// TIA Portal V17 program export: 9 tag tables, 0 data types, 25 data blocks, 98 code blocks (in call order from the OBs), 18 instance data blocks

VAR_GLOBAL   // PLC tag table "AIQ"
   IW100 AT %IW100 : Int;
   IW102 AT %IW102 : Int;
   IW104 AT %IW104 : Int;
   IW106 AT %IW106 : Int;
   IW108 AT %IW108 : Int;
   IW110 AT %IW110 : Int;
   IW112 AT %IW112 : Int;
   IW116 AT %IW116 : Int;
   IW118 AT %IW118 : Int;
   IW120 AT %IW120 : Int;
   IW122 AT %IW122 : Int;
   IW124 AT %IW124 : Int;
   IW126 AT %IW126 : Int;
   IW128 AT %IW128 : Int;
   IW130 AT %IW130 : Int;
   IW132 AT %IW132 : Int;
   IW134 AT %IW134 : Int;
   IW136 AT %IW136 : Int;
   IW138 AT %IW138 : Int;
   IW140 AT %IW140 : Int;
   IW142 AT %IW142 : Int;
   QW100 AT %QW100 : Int;
   QW102 AT %QW102 : Int;
   QW104 AT %QW104 : Int;
   QW106 AT %QW106 : Int;
   QW108 AT %QW108 : Int;
   QW110 AT %QW110 : Int;
   QW112 AT %QW112 : Int;
   QW114 AT %QW114 : Int;
   QW116 AT %QW116 : Int;
   QW118 AT %QW118 : Int;
   QW120 AT %QW120 : Int;
   QW122 AT %QW122 : Int;
   QW124 AT %QW124 : Int;
   QW126 AT %QW126 : Int;
   QW128 AT %QW128 : Int;
   QW130 AT %QW130 : Int;
   QW132 AT %QW132 : Int;
   QW134 AT %QW134 : Int;
   QW136 AT %QW136 : Int;
   QW138 AT %QW138 : Int;
   QW140 AT %QW140 : Int;
   QW142 AT %QW142 : Int;
   QW144 AT %QW144 : Int;
   QW146 AT %QW146 : Int;
   QW148 AT %QW148 : Int;
   QW150 AT %QW150 : Int;
   IW114 AT %IW114 : Int;
   IW144 AT %IW144 : Int;
   IW146 AT %IW146 : Int;
   IW148 AT %IW148 : Int;
   IW150 AT %IW150 : Int;
   IW152 AT %IW152 : Int;
   IW154 AT %IW154 : Int;
   IW156 AT %IW156 : Int;
   IW158 AT %IW158 : Int;
   IW160 AT %IW160 : Int;
   IW162 AT %IW162 : Int;
END_VAR

VAR_GLOBAL   // PLC tag table "AIQM"
   IWJF进风流量计 AT %MW600 : Int;
   IWJL进料流量 AT %MW602 : Int;
   IWJF进风压差变送器 AT %MW604 : Int;
   IWCF出风高效压差变送器 AT %MW606 : Int;
   IWBD布袋压差变送器 AT %MW608 : Int;
   IWSS输送高效压差变送器 AT %MW610 : Int;
   IWJL进料压力 AT %MW612 : Int;
   IWTN塔内压力 AT %MW614 : Int;
   IWGD管道压力变送器 AT %MW616 : Int;
   IWJD进氮压力 AT %MW618 : Int;
   IWFK放空比例反馈 AT %MW620 : Int;
   IWJF进风加热比例反馈 AT %MW622 : Int;
   IWHF回风加热比例反馈 AT %MW624 : Int;
   IWWH雾化油压 AT %MW626 : Int;
   IWYH氧含仪1 AT %MW628 : Int;
   IWYH氧含仪2 AT %MW630 : Int;
   IWYJ一级溶剂液位计 AT %MW632 : Int;
   IWEJ二级溶剂液位计 AT %MW634 : Int;
   IWCW除雾溶剂液位计 AT %MW636 : Int;
   IWSF送风机 AT %MW638 : Int;
   IWYF引风机 AT %MW640 : Int;
   IWLX离心雾化器 AT %MW642 : Int;
   IWJL进料泵 AT %MW644 : Int;
   QWSF送风机 AT %MW700 : Int;
   QWYF引风机 AT %MW702 : Int;
   QWLX离心雾化器 AT %MW704 : Int;
   QWJL进料泵 AT %MW706 : Int;
   QWFK放空比例调节阀 AT %MW708 : Int;
   QWJF进风加热比例调节阀 AT %MW710 : Int;
   QWHF回风加热比例调节阀 AT %MW712 : Int;
   IWFD阀岛气压 AT %MW646 : Int;
   IWQZ前置水罐液位计 AT %MW648 : Int;
   IWBY备用2 AT %MW650 : Int;
   IWBY备用3 AT %MW652 : Int;
   IWBY备用4 AT %MW654 : Int;
   IWBY备用5 AT %MW656 : Int;
   IWBY备用6 AT %MW658 : Int;
   IWBY备用7 AT %MW660 : Int;
   IWBY备用8 AT %MW662 : Int;
   IWBY备用9 AT %MW664 : Int;
END_VAR

VAR_GLOBAL   // PLC tag table "Alarm"
   A备用报警1 AT %M23.6 : Bool;
   AWK温控高温报警 AT %M37.7 : Bool;
   AKY空压低压信号 AT %M31.3 : Bool;
   ASS输送加热报警 AT %M34.7 : Bool;
   AWH雾化关报警 AT %M37.0 : Bool;
   AWH雾化开报警 AT %M37.1 : Bool;
   ABD布袋压差高报 AT %M20.2 : Bool;
   ABD布袋压差高高报 AT %M20.3 : Bool;
   AJF进风压差高高报 AT %M28.7 : Bool;
   AJF进风压差高报 AT %M28.6 : Bool;
   ATN塔内压力低报 AT %M36.4 : Bool;
   ATN塔内压力高报 AT %M36.6 : Bool;
   AJF进风温度高报 AT %M29.4 : Bool;
   AJF进风温度故障 AT %M29.3 : Bool;
   ACF出风温度高报 AT %M22.3 : Bool;
   ACF出风温度故障 AT %M22.1 : Bool;
   AWH雾化进氮低报 AT %M37.5 : Bool;
   AWQ尾气温度高报 AT %M38.1 : Bool;
   报警1 AT %MW20 : Word;
   ALD冷冻水关报警 AT %M31.4 : Bool;
   ACF出风温度过低 AT %M22.2 : Bool;
   AYH氧含量运行故障 AT %M39.2 : Bool;
   AJT急停报警 AT %M30.5 : Bool;
   报警2 AT %MW22 : Word;
   AJD进氮压力低报 AT %M27.3 : Bool;
   ATN塔内压力高高报 AT %M36.7 : Bool;
   AJF进风温度高高报 AT %M29.5 : Bool;
   ACF出风温度高高报 AT %M22.4 : Bool;
   ATN塔内压力低低报 AT %M36.3 : Bool;
   AWQ尾气温度高高报 AT %M38.2 : Bool;
   AGD管道压力高报 AT %M26.1 : Bool;
   AGD管道压力高高报 AT %M26.2 : Bool;
   AWQ尾气故障 AT %M38.0 : Bool;
   ALX离心雾化故障 AT %M31.7 : Bool;
   AJX机械温控故障 AT %M30.6 : Bool;
   AQT气体检测低报 AT %M32.4 : Bool;
   AQT气体检测低低报 AT %M32.3 : Bool;
   AWK温控未通信 AT %M37.6 : Bool;
   AHS回收罐1报警 AT %M26.7 : Bool;
   AHS回收罐2报警 AT %M27.0 : Bool;
   AJL进料泵故障报警 AT %M30.1 : Bool;
   AYF引风机报警 AT %M38.5 : Bool;
   AJB搅拌电机报警 AT %M27.1 : Bool;
   AQL气流雾化阀开报警 AT %M32.2 : Bool;
   AQL气流雾化阀关报警 AT %M32.1 : Bool;
   AYJ一级出料上阀开报警 AT %M39.6 : Bool;
   AYJ一级出料上阀关报警 AT %M39.5 : Bool;
   AYJ一级出料下阀开报警 AT %M40.0 : Bool;
   AYJ一级出料下阀关报警 AT %M39.7 : Bool;
   AEJ二级出料上阀开报警 AT %M24.2 : Bool;
   AEJ二级出料上阀关报警 AT %M24.1 : Bool;
   AEJ二级出料下阀开报警 AT %M24.4 : Bool;
   AEJ二级出料下阀关报警 AT %M24.3 : Bool;
   ACC除尘出料上阀开报警 AT %M21.5 : Bool;
   ACC除尘出料上阀关报警 AT %M21.4 : Bool;
   ACC除尘出料下阀开报警 AT %M21.7 : Bool;
   ACC除尘出料下阀关报警 AT %M21.6 : Bool;
   AKS开式排风隔断阀开报警 AT %M31.0 : Bool;
   AKS开式排风隔断阀关报警 AT %M30.7 : Bool;
   ABS闭式排风隔断阀开报警 AT %M21.1 : Bool;
   ABS闭式排风隔断阀关报警 AT %M21.0 : Bool;
   AKS开式进风隔断阀开报警 AT %M31.2 : Bool;
   AKS开式进风隔断阀关报警 AT %M31.1 : Bool;
   ABS闭式进风隔断阀开报警 AT %M21.3 : Bool;
   ABS闭式进风隔断阀关报警 AT %M21.2 : Bool;
   AYJ一级冷却水阀开报警 AT %M39.4 : Bool;
   AYJ一级冷却水阀关报警 AT %M39.3 : Bool;
   AEJ二级冷冻水阀开报警 AT %M24.0 : Bool;
   AEJ二级冷冻水阀关报警 AT %M23.7 : Bool;
   AYJ一级排液阀开报警 AT %M40.2 : Bool;
   AYJ一级排液阀关报警 AT %M40.1 : Bool;
   AEJ二级排液阀开报警 AT %M24.6 : Bool;
   AEJ二级排液阀关报警 AT %M24.5 : Bool;
   ACW除雾排液阀开报警 AT %M23.1 : Bool;
   ACW除雾排液阀关报警 AT %M23.0 : Bool;
   ARJ溶剂回收排放阀开报警 AT %M33.3 : Bool;
   ARJ溶剂回收排放阀关报警 AT %M33.2 : Bool;
   AXY泄压阀开报警 AT %M38.4 : Bool;
   AXY泄压阀关报警 AT %M38.3 : Bool;
   AJF进风冷却水阀开报警 AT %M28.2 : Bool;
   AJF进风冷却水阀关报警 AT %M28.1 : Bool;
   ASS输送进风阀开报警 AT %M35.4 : Bool;
   ASS输送进风阀关报警 AT %M35.3 : Bool;
   ASS输送出料上阀开报警 AT %M34.4 : Bool;
   ASS输送出料上阀关报警 AT %M34.3 : Bool;
   ASS输送出料下阀开报警 AT %M34.6 : Bool;
   ASS输送出料下阀关报警 AT %M34.5 : Bool;
   ATD塔顶清洗球阀开报警 AT %M36.2 : Bool;
   ATD塔顶清洗球阀关报警 AT %M36.1 : Bool;
   AQX清洗伸缩气缸开报警 AT %M32.6 : Bool;
   AQX清洗伸缩气缸关报警 AT %M32.5 : Bool;
   ABD补氮阀开报警 AT %M20.5 : Bool;
   ABD补氮阀关报警 AT %M20.4 : Bool;
   AJD进氮阀开报警 AT %M27.6 : Bool;
   AJD进氮阀关报警 AT %M27.5 : Bool;
   ASF送风机报警 AT %M33.7 : Bool;
   AJF进风保护温度报警 AT %M27.7 : Bool;
   ASS输送保护温度报警 AT %M34.2 : Bool;
   ABP爆破片1反馈报警 AT %M20.6 : Bool;
   ABP爆破片2反馈报警 AT %M20.7 : Bool;
   ASN室内排水开反馈报警 AT %M34.1 : Bool;
   ASN室内排水关反馈报警 AT %M34.0 : Bool;
   ADJ电加热报警 AT %M23.5 : Bool;
   AWH雾化油压低报 AT %M37.3 : Bool;
   AWH雾化油压低低报 AT %M37.2 : Bool;
   AJD进氮压力低低报 AT %M27.2 : Bool;
   AFD阀导气压低报 AT %M25.3 : Bool;
   AFD阀导气压低低报 AT %M25.2 : Bool;
   AJF进风压差低报 AT %M28.4 : Bool;
   ACF出风高效高报 AT %M22.6 : Bool;
   ACF出风高效高高报 AT %M22.7 : Bool;
   ACF出风高效低报 AT %M22.5 : Bool;
   ASS输送高效高报 AT %M35.7 : Bool;
   ASS输送高效高高报 AT %M36.0 : Bool;
   ASF输送高效低报 AT %M33.6 : Bool;
   AHF回风温度高报 AT %M26.5 : Bool;
   AHF回风温度高高报 AT %M26.6 : Bool;
   AJF进风冷却水流量低报警 AT %M28.0 : Bool;
   ALD冷冻水流量低报警 AT %M31.5 : Bool;
   ALQ冷却水流量低报警 AT %M31.6 : Bool;
   ABD布袋压差低报 AT %M20.0 : Bool;
   AJF进风流量计故障 AT %M29.2 : Bool;
   AJL进料流量故障 AT %M30.4 : Bool;
   AJF进风压差变送器故障 AT %M28.5 : Bool;
   ACF出风压差变送器故障 AT %M22.0 : Bool;
   ABD布袋压差变送器故障 AT %M20.1 : Bool;
   ASS输送高效压差变送器故障 AT %M35.6 : Bool;
   AJL进料压力故障 AT %M29.6 : Bool;
   ATN塔内压力故障 AT %M36.5 : Bool;
   AGD管道压力变送器故障 AT %M26.0 : Bool;
   AJD进氮压力故障 AT %M27.4 : Bool;
   AFK放空比例反馈故障 AT %M25.7 : Bool;
   AJF进风加热比例反馈故障 AT %M28.3 : Bool;
   AHF回风加热比例反馈故障 AT %M26.3 : Bool;
   AWH雾化油压故障 AT %M37.4 : Bool;
   AYH氧含仪1故障 AT %M38.6 : Bool;
   AYH氧含仪2故障 AT %M38.7 : Bool;
   AYJ一级溶剂液位计故障 AT %M40.5 : Bool;
   AEJ二级溶剂液位计故障 AT %M25.1 : Bool;
   ACW除雾溶剂液位计故障 AT %M23.4 : Bool;
   AFD阀岛气压故障报警 AT %M25.6 : Bool;
   AJL进料压力高报 AT %M29.7 : Bool;
   AJL进料压力高高报 AT %M30.0 : Bool;
   ASS输送温度高高报 AT %M35.2 : Bool;
   ASS输送温度高报 AT %M35.1 : Bool;
   ASS输送温度故障报警 AT %M35.0 : Bool;
   AHF回风温度故障报警 AT %M26.4 : Bool;
   ASS输送高效低报 AT %M35.5 : Bool;
   AYJ一级液位计高报 AT %M40.3 : Bool;
   AYJ一级液位计高高报 AT %M40.4 : Bool;
   AEJ二级液位计高报 AT %M24.7 : Bool;
   AEJ二级液位计高高报 AT %M25.0 : Bool;
   ACW除雾液位计高报 AT %M23.2 : Bool;
   ACW除雾液位计高高报 AT %M23.3 : Bool;
   AFD阀岛气压低报 AT %M25.5 : Bool;
   AFD阀岛气压低低报 AT %M25.4 : Bool;
   APY排液流量低报警 AT %M32.0 : Bool;
   ASF输送风机故障报警 AT %M33.5 : Bool;
   ASF输送加热故障报警 AT %M33.4 : Bool;
   AYH氧含仪高报 AT %M39.0 : Bool;
   AYH氧含仪高高报 AT %M39.1 : Bool;
   AJF进风流量低低报 AT %M29.0 : Bool;
   AJF进风流量低报 AT %M29.1 : Bool;
   AQZ前置液位低报 AT %M33.0 : Bool;
   AQZ前置液位低低报 AT %M32.7 : Bool;
   AQZ前置液位计故障 AT %M33.1 : Bool;
   AJL进料流量低报 AT %M30.3 : Bool;
   AJL进料流量低低报 AT %M30.2 : Bool;
   报警3 AT %MW24 : Word;
   报警4 AT %MW26 : Word;
   报警5 AT %MW28 : Word;
   报警6 AT %MW30 : Word;
   报警7 AT %MW32 : Word;
   报警8 AT %MW34 : Word;
   报警9 AT %MW36 : Word;
   报警10 AT %MW38 : Word;
   报警11 AT %MW40 : Word;
   报警12 AT %MW42 : Word;
   AKS开式自动自检不通过 AT %M40.6 : Bool;
   ACIP缺水报警 AT %M40.7 : Bool;
   ARJ溶剂排液泵开报警 AT %M41.0 : Bool;
   ARJ溶剂排液泵关报警 AT %M41.1 : Bool;
END_VAR

VAR_GLOBAL   // PLC tag table "COM"
   CSJ时间更改 AT %M50.2 : Bool;
   CBD本地读 AT %MW54 : Int;
   CJF进温SW写 AT %MW56 : Int;
   CJB搅拌1温SW写 AT %MW58 : Int;
   CJB搅拌2温SW写 AT %MW60 : Int;
END_VAR

VAR_GLOBAL   // PLC tag table "IO"
   "I0.0" AT %I0.0 : Bool;
   "I0.1" AT %I0.1 : Bool;
   "I0.2" AT %I0.2 : Bool;
   "I0.3" AT %I0.3 : Bool;
   "I0.4" AT %I0.4 : Bool;
   "I0.5" AT %I0.5 : Bool;
   "I0.6" AT %I0.6 : Bool;
   "I0.7" AT %I0.7 : Bool;
   "I1.0" AT %I1.0 : Bool;
   "I1.1" AT %I1.1 : Bool;
   "I2.0" AT %I2.0 : Bool;
   "I2.1" AT %I2.1 : Bool;
   "I2.2" AT %I2.2 : Bool;
   "I2.3" AT %I2.3 : Bool;
   "I2.4" AT %I2.4 : Bool;
   "I2.5" AT %I2.5 : Bool;
   "I2.6" AT %I2.6 : Bool;
   "I2.7" AT %I2.7 : Bool;
   "I3.0" AT %I3.0 : Bool;
   "I3.1" AT %I3.1 : Bool;
   "I3.2" AT %I3.2 : Bool;
   "I3.3" AT %I3.3 : Bool;
   "I3.4" AT %I3.4 : Bool;
   "I3.5" AT %I3.5 : Bool;
   "I3.6" AT %I3.6 : Bool;
   "I3.7" AT %I3.7 : Bool;
   "I4.0" AT %I4.0 : Bool;
   "I4.1" AT %I4.1 : Bool;
   "I4.2" AT %I4.2 : Bool;
   "I4.3" AT %I4.3 : Bool;
   "I4.4" AT %I4.4 : Bool;
   "I4.5" AT %I4.5 : Bool;
   "I4.6" AT %I4.6 : Bool;
   "I4.7" AT %I4.7 : Bool;
   "I5.0" AT %I5.0 : Bool;
   "I5.1" AT %I5.1 : Bool;
   "I5.2" AT %I5.2 : Bool;
   "I5.3" AT %I5.3 : Bool;
   "I5.4" AT %I5.4 : Bool;
   "I5.5" AT %I5.5 : Bool;
   "I5.6" AT %I5.6 : Bool;
   "I5.7" AT %I5.7 : Bool;
   "Q0.1" AT %Q0.1 : Bool;
   "Q0.2" AT %Q0.2 : Bool;
   "Q0.3" AT %Q0.3 : Bool;
   "Q0.4" AT %Q0.4 : Bool;
   "Q0.5" AT %Q0.5 : Bool;
   "Q0.6" AT %Q0.6 : Bool;
   "Q0.7" AT %Q0.7 : Bool;
   "Q1.0" AT %Q1.0 : Bool;
   "Q1.1" AT %Q1.1 : Bool;
   "Q1.2" AT %Q1.2 : Bool;
   "Q1.3" AT %Q1.3 : Bool;
   "Q1.4" AT %Q1.4 : Bool;
   "Q1.5" AT %Q1.5 : Bool;
   "Q3.0" AT %Q3.0 : Bool;
   "Q3.1" AT %Q3.1 : Bool;
   "Q3.2" AT %Q3.2 : Bool;
   "Q3.3" AT %Q3.3 : Bool;
   "Q3.4" AT %Q3.4 : Bool;
   "Q3.5" AT %Q3.5 : Bool;
   "Q3.6" AT %Q3.6 : Bool;
   "Q3.7" AT %Q3.7 : Bool;
   "Q4.0" AT %Q4.0 : Bool;
   "Q4.1" AT %Q4.1 : Bool;
   "Q4.2" AT %Q4.2 : Bool;
   "Q4.3" AT %Q4.3 : Bool;
   "Q4.4" AT %Q4.4 : Bool;
   "Q4.5" AT %Q4.5 : Bool;
   "Q4.6" AT %Q4.6 : Bool;
   "Q4.7" AT %Q4.7 : Bool;
   "Q5.0" AT %Q5.0 : Bool;
   "Q5.1" AT %Q5.1 : Bool;
   "Q5.2" AT %Q5.2 : Bool;
   "Q5.3" AT %Q5.3 : Bool;
   "Q5.4" AT %Q5.4 : Bool;
   "Q0.0" AT %Q0.0 : Bool;
   "I1.2" AT %I1.2 : Bool;
   "I1.3" AT %I1.3 : Bool;
   "I1.4" AT %I1.4 : Bool;
   "I1.5" AT %I1.5 : Bool;
   "Q5.5" AT %Q5.5 : Bool;
   "Q1.6" AT %Q1.6 : Bool;
   "Q1.7" AT %Q1.7 : Bool;
   "I1.6" AT %I1.6 : Bool;
   "I1.7" AT %I1.7 : Bool;
   "Q5.6" AT %Q5.6 : Bool;
   "Q5.7" AT %Q5.7 : Bool;
   "Q6.0" AT %Q6.0 : Bool;
   "Q6.1" AT %Q6.1 : Bool;
   "Q6.2" AT %Q6.2 : Bool;
   "Q6.3" AT %Q6.3 : Bool;
   "Q6.4" AT %Q6.4 : Bool;
   "Q6.5" AT %Q6.5 : Bool;
   "Q6.6" AT %Q6.6 : Bool;
   "Q6.7" AT %Q6.7 : Bool;
   "Q7.0" AT %Q7.0 : Bool;
   "Q7.1" AT %Q7.1 : Bool;
   "Q7.2" AT %Q7.2 : Bool;
   "Q7.3" AT %Q7.3 : Bool;
   "Q7.4" AT %Q7.4 : Bool;
   "Q7.5" AT %Q7.5 : Bool;
   "Q7.6" AT %Q7.6 : Bool;
   "Q7.7" AT %Q7.7 : Bool;
   "Q8.0" AT %Q8.0 : Bool;
   "Q8.1" AT %Q8.1 : Bool;
   "Q8.2" AT %Q8.2 : Bool;
   "Q8.3" AT %Q8.3 : Bool;
   "Q8.4" AT %Q8.4 : Bool;
   "Q8.5" AT %Q8.5 : Bool;
   "Q8.6" AT %Q8.6 : Bool;
   "Q8.7" AT %Q8.7 : Bool;
   "Q9.0" AT %Q9.0 : Bool;
   "Q9.1" AT %Q9.1 : Bool;
   "Q9.2" AT %Q9.2 : Bool;
   "Q9.3" AT %Q9.3 : Bool;
   "Q9.4" AT %Q9.4 : Bool;
   "Q9.5" AT %Q9.5 : Bool;
   "Q9.6" AT %Q9.6 : Bool;
   "Q9.7" AT %Q9.7 : Bool;
   "Q10.0" AT %Q10.0 : Bool;
   "Q10.1" AT %Q10.1 : Bool;
   "Q10.2" AT %Q10.2 : Bool;
   "Q10.3" AT %Q10.3 : Bool;
   "I6.0" AT %I6.0 : Bool;
   "I6.1" AT %I6.1 : Bool;
   "I6.2" AT %I6.2 : Bool;
   "I6.3" AT %I6.3 : Bool;
   "I6.4" AT %I6.4 : Bool;
   "I6.5" AT %I6.5 : Bool;
   "I6.6" AT %I6.6 : Bool;
   "I6.7" AT %I6.7 : Bool;
   "I7.0" AT %I7.0 : Bool;
   "I7.1" AT %I7.1 : Bool;
   "I7.2" AT %I7.2 : Bool;
   "I7.3" AT %I7.3 : Bool;
   "I7.4" AT %I7.4 : Bool;
   "I7.5" AT %I7.5 : Bool;
   "I7.6" AT %I7.6 : Bool;
   "I7.7" AT %I7.7 : Bool;
   "Q10.4" AT %Q10.4 : Bool;
   "Q10.5" AT %Q10.5 : Bool;
   "Q10.6" AT %Q10.6 : Bool;
   "Q10.7" AT %Q10.7 : Bool;
   "Q11.0" AT %Q11.0 : Bool;
   "Q11.1" AT %Q11.1 : Bool;
   "Q11.2" AT %Q11.2 : Bool;
   "Q11.3" AT %Q11.3 : Bool;
   "Q11.4" AT %Q11.4 : Bool;
   "Q11.5" AT %Q11.5 : Bool;
   "Q11.6" AT %Q11.6 : Bool;
   "Q11.7" AT %Q11.7 : Bool;
   "Q12.0" AT %Q12.0 : Bool;
   "Q12.1" AT %Q12.1 : Bool;
   "Q12.2" AT %Q12.2 : Bool;
   "Q12.3" AT %Q12.3 : Bool;
   "Q12.4" AT %Q12.4 : Bool;
   "Q12.5" AT %Q12.5 : Bool;
   "Q12.6" AT %Q12.6 : Bool;
   "Q12.7" AT %Q12.7 : Bool;
   "Q13.0" AT %Q13.0 : Bool;
   "Q13.1" AT %Q13.1 : Bool;
   "Q13.2" AT %Q13.2 : Bool;
   "Q13.3" AT %Q13.3 : Bool;
   "Q13.4" AT %Q13.4 : Bool;
   "Q13.5" AT %Q13.5 : Bool;
   "Q13.6" AT %Q13.6 : Bool;
   "Q13.7" AT %Q13.7 : Bool;
   "Q14.0" AT %Q14.0 : Bool;
   "Q14.1" AT %Q14.1 : Bool;
   "Q14.2" AT %Q14.2 : Bool;
   "Q14.3" AT %Q14.3 : Bool;
   "Q14.4" AT %Q14.4 : Bool;
   "Q14.5" AT %Q14.5 : Bool;
   "Q14.6" AT %Q14.6 : Bool;
   "Q14.7" AT %Q14.7 : Bool;
   "Q15.0" AT %Q15.0 : Bool;
   "Q15.1" AT %Q15.1 : Bool;
   "Q15.2" AT %Q15.2 : Bool;
   "Q15.3" AT %Q15.3 : Bool;
   "Q15.4" AT %Q15.4 : Bool;
   "Q15.5" AT %Q15.5 : Bool;
   "Q15.6" AT %Q15.6 : Bool;
   "Q15.7" AT %Q15.7 : Bool;
   "Q16.0" AT %Q16.0 : Bool;
   "Q16.1" AT %Q16.1 : Bool;
   "Q16.2" AT %Q16.2 : Bool;
   "Q16.3" AT %Q16.3 : Bool;
   "Q16.4" AT %Q16.4 : Bool;
   "Q16.5" AT %Q16.5 : Bool;
   "Q16.6" AT %Q16.6 : Bool;
   "Q16.7" AT %Q16.7 : Bool;
   "Q17.0" AT %Q17.0 : Bool;
   "Q17.1" AT %Q17.1 : Bool;
   "Q17.2" AT %Q17.2 : Bool;
   "Q17.3" AT %Q17.3 : Bool;
   "Q17.4" AT %Q17.4 : Bool;
   "Q17.5" AT %Q17.5 : Bool;
   "Q17.6" AT %Q17.6 : Bool;
   "Q17.7" AT %Q17.7 : Bool;
   "Q18.0" AT %Q18.0 : Bool;
   "Q18.1" AT %Q18.1 : Bool;
   "Q18.2" AT %Q18.2 : Bool;
   "Q18.3" AT %Q18.3 : Bool;
   "Q18.4" AT %Q18.4 : Bool;
   "Q18.5" AT %Q18.5 : Bool;
   "Q18.6" AT %Q18.6 : Bool;
   "Q18.7" AT %Q18.7 : Bool;
   "Q19.0" AT %Q19.0 : Bool;
   "Q19.1" AT %Q19.1 : Bool;
   "Q19.2" AT %Q19.2 : Bool;
   "Q19.3" AT %Q19.3 : Bool;
   "Q19.4" AT %Q19.4 : Bool;
   "Q19.5" AT %Q19.5 : Bool;
   "Q19.6" AT %Q19.6 : Bool;
   "Q19.7" AT %Q19.7 : Bool;
   "Q20.0" AT %Q20.0 : Bool;
   "Q20.1" AT %Q20.1 : Bool;
   "Q20.2" AT %Q20.2 : Bool;
   "Q20.3" AT %Q20.3 : Bool;
   "Q20.4" AT %Q20.4 : Bool;
   "Q20.5" AT %Q20.5 : Bool;
   "Q2.0" AT %Q2.0 : Bool;
   "Q2.1" AT %Q2.1 : Bool;
   "Q2.2" AT %Q2.2 : Bool;
   "Q2.3" AT %Q2.3 : Bool;
   "Q2.4" AT %Q2.4 : Bool;
   "Q2.5" AT %Q2.5 : Bool;
   "Q2.6" AT %Q2.6 : Bool;
   "Q2.7" AT %Q2.7 : Bool;
END_VAR

VAR_GLOBAL   // PLC tag table "IOM"
   QSF送风机 AT %M300.0 : Bool;
   QSF送风机风扇 AT %M300.1 : Bool;
   QDJ电加热器 AT %M301.1 : Bool;
   QSS输送风机 AT %M301.2 : Bool;
   QSS输送加热器 AT %M301.3 : Bool;
   QYF引风机 AT %M300.2 : Bool;
   QYF引风机风扇 AT %M300.3 : Bool;
   QLX离心雾化 AT %M300.4 : Bool;
   QLX离心雾化风扇 AT %M300.5 : Bool;
   QLX离心雾化油泵 AT %M300.6 : Bool;
   QJL进料泵 AT %M300.7 : Bool;
   QJL进料泵风扇 AT %M301.0 : Bool;
   QFM蜂鸣器 AT %M301.4 : Bool;
   QZS指示灯 AT %M301.5 : Bool;
   QYS钥匙开关 AT %M301.6 : Bool;
   QZM照明灯 AT %M301.7 : Bool;
   QPH平衡比例调节阀 AT %M302.0 : Bool;
   QCC除尘脉冲 AT %M302.1 : Bool;
   QJF进风蒸汽比例调节阀 AT %M302.2 : Bool;
   QHF回风蒸汽调节阀 AT %M302.3 : Bool;
   QBY备用1 AT %M302.4 : Bool;
   QBY备用2 AT %M302.5 : Bool;
   QBY备用3 AT %M302.6 : Bool;
   QBY备用4 AT %M302.7 : Bool;
   QXY泄压阀 AT %M303.0 : Bool;
   QJF进风冷却水阀 AT %M303.1 : Bool;
   QSS输送进风阀 AT %M303.2 : Bool;
   QQL气流雾化阀 AT %M303.3 : Bool;
   QKS开式排风隔断阀 AT %M303.4 : Bool;
   QBS闭式排风隔断阀 AT %M303.5 : Bool;
   QKS开式进风隔断阀 AT %M303.6 : Bool;
   QBS闭式进风隔断阀 AT %M303.7 : Bool;
   QYJ一级冷却水阀 AT %M304.0 : Bool;
   QEJ二级冷冻水阀 AT %M304.1 : Bool;
   QYJ一级排液阀 AT %M304.2 : Bool;
   QEJ二级排液阀 AT %M304.3 : Bool;
   QCW除雾排液阀 AT %M304.4 : Bool;
   QRJ溶剂回收排放阀 AT %M304.5 : Bool;
   QZT主塔气锤1 AT %M304.6 : Bool;
   QZT主塔气锤2 AT %M304.7 : Bool;
   QZT主塔气锤3 AT %M305.0 : Bool;
   QZT主塔气锤4 AT %M305.1 : Bool;
   QASA室内回水阀 AT %M305.2 : Bool;
   QYJ一级缓存振荡器 AT %M305.3 : Bool;
   QASA室外回水阀 AT %M305.4 : Bool;
   QEJ二级缓存震荡器 AT %M305.5 : Bool;
   QCC除尘气锤1 AT %M305.6 : Bool;
   QCC除尘气锤2 AT %M305.7 : Bool;
   QCC除尘缓存震荡器 AT %M306.0 : Bool;
   QRJ溶剂排液泵进阀 AT %M306.1 : Bool;
   QSN室内清洗总阀 AT %M306.2 : Bool;
   QBD补氮阀 AT %M306.3 : Bool;
   QJD进氮阀 AT %M306.4 : Bool;
   QJF进风蒸汽开关阀 AT %M306.5 : Bool;
   QJF进风蒸汽排水阀 AT %M306.6 : Bool;
   QLG料罐清洗阀 AT %M306.7 : Bool;
   QQX清洗溶剂出阀 AT %M307.0 : Bool;
   QWL物料进阀 AT %M307.1 : Bool;
   QYJ一级出料上阀 AT %M307.2 : Bool;
   QYJ一级出料下阀 AT %M307.3 : Bool;
   QEJ二级出料上阀 AT %M307.4 : Bool;
   QEJ二级出料下阀 AT %M307.5 : Bool;
   QCC除尘出料上阀 AT %M307.6 : Bool;
   QCC除尘出料下阀 AT %M307.7 : Bool;
   QHF回风蒸汽开关阀 AT %M308.0 : Bool;
   QHF回风蒸汽排水阀 AT %M308.1 : Bool;
   QSS输送出料上阀 AT %M308.2 : Bool;
   QSS输送出料下阀 AT %M308.3 : Bool;
   QTD塔顶清洗球阀 AT %M308.4 : Bool;
   QQG气缸升降阀 AT %M308.5 : Bool;
   QZT主塔清洗进水阀 AT %M308.6 : Bool;
   QXF旋风管道清洗阀 AT %M308.7 : Bool;
   QYJ一级旋风清洗阀 AT %M309.0 : Bool;
   QEJ二级旋风清洗阀 AT %M309.1 : Bool;
   QCC除尘管道清洗阀 AT %M309.2 : Bool;
   QCC除尘清洗阀 AT %M309.3 : Bool;
   QSS输送管路清洗阀 AT %M309.4 : Bool;
   QLC料仓清洗阀 AT %M309.5 : Bool;
   QJR加热清洗阀 AT %M309.6 : Bool;
   QWK蜗壳清洗阀 AT %M309.7 : Bool;
   QCF出风高效清洗阀 AT %M310.0 : Bool;
   QZT主塔排水阀 AT %M310.1 : Bool;
   QSS输送管路排水阀 AT %M310.2 : Bool;
   QLC料仓清洗排水阀 AT %M310.3 : Bool;
   QSF送风机清洗阀 AT %M310.4 : Bool;
   QYF引风机清洗阀 AT %M310.5 : Bool;
   QYJ一级冷凝清洗阀 AT %M310.6 : Bool;
   QEJ二级冷凝清洗阀 AT %M310.7 : Bool;
   QSF送风机排水阀 AT %M311.0 : Bool;
   QYF引风机排水阀 AT %M311.1 : Bool;
   ISF送风机 AT %M350.0 : Bool;
   IYF引风机 AT %M350.1 : Bool;
   ILX离心雾化器 AT %M350.2 : Bool;
   IJL进料泵 AT %M350.3 : Bool;
   IDJ电加热 AT %M350.4 : Bool;
   ISF输送风机 AT %M350.5 : Bool;
   ISF输送加热 AT %M350.6 : Bool;
   IJT急停 AT %M350.7 : Bool;
   ILQ冷却水流量 AT %M351.0 : Bool;
   ILD冷冻水流量 AT %M351.1 : Bool;
   IJF进风冷却水流量 AT %M351.2 : Bool;
   IPY排液流量 AT %M351.3 : Bool;
   IBD补氮阀开反馈 AT %M351.4 : Bool;
   IBD补氮阀关反馈 AT %M351.5 : Bool;
   IJD进氮阀开反馈 AT %M351.6 : Bool;
   IJD进氮阀关反馈 AT %M351.7 : Bool;
   IXY泄压阀开反馈 AT %M352.0 : Bool;
   IXY泄压阀关反馈 AT %M352.1 : Bool;
   IQL气流雾化阀开反馈 AT %M352.2 : Bool;
   IQL气流雾化阀关反馈 AT %M352.3 : Bool;
   ISF输送进风阀开反馈 AT %M352.4 : Bool;
   ISF输送进风阀关反馈 AT %M352.5 : Bool;
   IKS开式排风隔断阀开反馈 AT %M352.6 : Bool;
   IKS开式排风隔断阀关反馈 AT %M352.7 : Bool;
   IBS闭式排风隔断阀开反馈 AT %M353.0 : Bool;
   IBS闭式排风隔断阀关反馈 AT %M353.1 : Bool;
   IKS开式进风隔断阀开反馈 AT %M353.2 : Bool;
   IKS开式进风隔断阀关反馈 AT %M353.3 : Bool;
   IBS闭式进风隔断阀开反馈 AT %M353.4 : Bool;
   IBS闭式进风隔断阀关反馈 AT %M353.5 : Bool;
   IYJ一级冷却水阀开反馈 AT %M353.6 : Bool;
   IYJ一级冷却水阀关反馈 AT %M353.7 : Bool;
   IEJ二级冷冻水阀开反馈 AT %M354.0 : Bool;
   IEJ二级冷冻水阀关反馈 AT %M354.1 : Bool;
   IYJ一级排液阀开反馈 AT %M354.2 : Bool;
   IYJ一级排液阀关反馈 AT %M354.3 : Bool;
   IEJ二级排液阀开反馈 AT %M354.4 : Bool;
   IEJ二级排液阀关反馈 AT %M354.5 : Bool;
   ICW除雾排液阀开反馈 AT %M354.6 : Bool;
   ICW除雾排液阀关反馈 AT %M354.7 : Bool;
   IRJ溶剂回收排放阀开反馈 AT %M355.0 : Bool;
   IRJ溶剂回收排放阀关反馈 AT %M355.1 : Bool;
   IJF进风冷却水阀开反馈 AT %M355.2 : Bool;
   IJF进风冷却水阀关反馈 AT %M355.3 : Bool;
   ITD塔顶清洗球阀开反馈 AT %M355.4 : Bool;
   ITD塔顶清洗球阀关反馈 AT %M355.5 : Bool;
   IQX清洗伸缩气缸降反馈 AT %M355.6 : Bool;
   IQX清洗伸缩气缸升反馈 AT %M355.7 : Bool;
   QRS热水洗请求 AT %M311.2 : Bool;
   QRJ溶剂洗 AT %M311.3 : Bool;
   QBY备用7 AT %M311.4 : Bool;
   QSN室内排水隔膜泵 AT %M311.5 : Bool;
   QRJ溶剂排液泵 AT %M311.6 : Bool;
   QBY备用10 AT %M311.7 : Bool;
   QBY备用11 AT %M312.0 : Bool;
   QBY备用12 AT %M312.1 : Bool;
   QBY备用13 AT %M312.2 : Bool;
   QBY备用14 AT %M312.3 : Bool;
   QBY备用15 AT %M312.4 : Bool;
   QBY备用16 AT %M312.5 : Bool;
   QBY备用17 AT %M312.6 : Bool;
   QBY备用18 AT %M312.7 : Bool;
   QBY备用19 AT %M313.0 : Bool;
   QBY备用20 AT %M313.1 : Bool;
   QQG气缸升 AT %M313.2 : Bool;
   QQG气缸降 AT %M313.3 : Bool;
   QBD布袋振打1 AT %M313.4 : Bool;
   QSB设备振打 AT %M313.5 : Bool;
   QBD布袋振打3 AT %M313.6 : Bool;
   QBD布袋振打4 AT %M313.7 : Bool;
   QYH氧含仪隔断阀 AT %M314.0 : Bool;
   QHS回水隔断阀1 AT %M314.1 : Bool;
   IJF进风保护温度 AT %M356.0 : Bool;
   ISS输送保护温度 AT %M356.1 : Bool;
   IBP爆破片1反馈 AT %M356.2 : Bool;
   IBP爆破片2反馈 AT %M356.3 : Bool;
   ISN室内排水开反馈 AT %M356.4 : Bool;
   ISN室内排水关反馈 AT %M356.5 : Bool;
   IRJ溶剂排液泵开反馈 AT %M356.6 : Bool;
   IRJ溶剂排液泵关反馈 AT %M356.7 : Bool;
   QXT心跳发送信号 AT %M314.2 : Bool;
   QCS纯水洗请求 AT %M314.3 : Bool;
   QJS碱水洗请求 AT %M314.4 : Bool;
   QRJ溶剂请求 AT %M314.5 : Bool;
   QYG压干请求 AT %M314.6 : Bool;
   QQZ前置水阀 AT %M314.7 : Bool;
   QYJ一级旋风振打锤 AT %M315.0 : Bool;
   QEJ二级旋风振打锤 AT %M315.1 : Bool;
   QYJ一级旋风振荡器 AT %M315.2 : Bool;
   QCIP启动 AT %M315.3 : Bool;
   QGS供水泵启动 AT %M315.4 : Bool;
   QZS注射水洗 AT %M315.5 : Bool;
   QSJ水进程泵 AT %M315.6 : Bool;
   QRJ溶剂进程泵 AT %M315.7 : Bool;
   QQS缺水状态 AT %M316.0 : Bool;
   QRC热纯自动洗 AT %M316.1 : Bool;
END_VAR

VAR_GLOBAL   // PLC tag table "M"
   MMC脉冲反吹 AT %M400.0 : Bool;
   MJF进温自整定 AT %M400.1 : Bool;
   MSF送风机 AT %M400.2 : Bool;
   MSF送风机风扇 AT %M400.3 : Bool;
   MDJ电加热器 AT %M400.4 : Bool;
   MLX离心雾化 AT %M400.5 : Bool;
   MLX离心雾化风扇 AT %M400.6 : Bool;
   MLX离心雾化油泵 AT %M400.7 : Bool;
   MJL进料泵 AT %M401.0 : Bool;
   MJL进料泵风扇 AT %M401.1 : Bool;
   MYF引风机 AT %M401.2 : Bool;
   MYF引风机风扇 AT %M401.3 : Bool;
   MSF输送风机 AT %M401.4 : Bool;
   MSF输送加热器 AT %M401.5 : Bool;
   MRJ溶剂排液泵 AT %M401.6 : Bool;
   MCC除尘脉冲 AT %M401.7 : Bool;
   MFM蜂鸣器 AT %M402.0 : Bool;
   MZS指示灯 AT %M402.1 : Bool;
   MYS钥匙开关 AT %M402.2 : Bool;
   MQX清洗溶剂罐进氮阀 AT %M402.3 : Bool;
   MBD补氮阀 AT %M402.4 : Bool;
   MJD进氮阀 AT %M402.5 : Bool;
   MJF进风蒸汽开关阀 AT %M402.6 : Bool;
   MJF进风蒸汽比例调节阀 AT %M402.7 : Bool;
   MJF进风蒸汽排水阀 AT %M403.0 : Bool;
   MQX清洗溶剂进阀 AT %M403.1 : Bool;
   MQX清洗溶剂出阀 AT %M403.2 : Bool;
   MWL物料进阀 AT %M403.3 : Bool;
   MYJ一级出料上阀 AT %M403.4 : Bool;
   MYJ一级出料下阀 AT %M403.5 : Bool;
   MEJ二级出料上阀 AT %M403.6 : Bool;
   MEJ二级出料下阀 AT %M403.7 : Bool;
   MCC除尘出料上阀 AT %M404.0 : Bool;
   MCC除尘出料下阀 AT %M404.1 : Bool;
   MKS开式排风隔断阀 AT %M404.2 : Bool;
   MBS闭式排风隔断阀 AT %M404.3 : Bool;
   MKS开式进风隔断阀 AT %M404.4 : Bool;
   MBS闭式进风隔断阀 AT %M404.5 : Bool;
   MYJ一级冷却水阀 AT %M404.6 : Bool;
   MYJ二级冷冻水阀 AT %M404.7 : Bool;
   MYJ一级排液阀 AT %M405.0 : Bool;
   MEJ二级排液阀 AT %M405.1 : Bool;
   MCW除雾排液阀 AT %M405.2 : Bool;
   MRJ溶剂回收排放阀 AT %M405.3 : Bool;
   MHF回风蒸汽开关阀 AT %M405.4 : Bool;
   MHF回风蒸汽调节阀 AT %M405.5 : Bool;
   MHF回风蒸汽排水阀 AT %M405.6 : Bool;
   MXY泄压阀 AT %M405.7 : Bool;
   MPH平衡比例调节阀 AT %M406.0 : Bool;
   MJF进风冷却水阀 AT %M406.1 : Bool;
   MSS输送进风阀 AT %M406.2 : Bool;
   MSS输送出料上阀 AT %M406.3 : Bool;
   MSS输送出料下阀 AT %M406.4 : Bool;
   MQL气流雾化阀 AT %M406.5 : Bool;
   MZT主塔气锤 AT %M406.6 : Bool;
   MYJ一级旋风气锤 AT %M406.7 : Bool;
   MYJ一级缓存振荡器 AT %M407.0 : Bool;
   MEJ二级旋风气锤 AT %M407.1 : Bool;
   MEJ二级缓存震荡器 AT %M407.2 : Bool;
   MCC除尘气锤 AT %M407.3 : Bool;
   MCC除尘缓存震荡器 AT %M407.4 : Bool;
   MTD塔顶清洗球阀 AT %M407.5 : Bool;
   MQG气缸升降阀 AT %M407.6 : Bool;
   MZT主塔清洗进水阀 AT %M407.7 : Bool;
   MXF旋风管道清洗阀 AT %M408.0 : Bool;
   MYJ一级旋风清洗阀 AT %M408.1 : Bool;
   MEJ二级旋风清洗阀 AT %M408.2 : Bool;
   MCC除尘管道清洗阀 AT %M408.3 : Bool;
   MCC除尘清洗阀 AT %M408.4 : Bool;
   MSS输送管路清洗阀 AT %M408.5 : Bool;
   MLC料仓清洗阀 AT %M408.6 : Bool;
   MJR加热清洗阀 AT %M408.7 : Bool;
   MWK蜗壳清洗阀 AT %M409.0 : Bool;
   MCF出风高效清洗阀 AT %M409.1 : Bool;
   MZT主塔排水阀 AT %M409.2 : Bool;
   MSS输送管路排水阀 AT %M409.3 : Bool;
   MLC料仓清洗排水阀 AT %M409.4 : Bool;
   MSF送风机清洗阀 AT %M409.5 : Bool;
   MYF引风机清洗阀 AT %M409.6 : Bool;
   MYJ一级冷凝清洗阀 AT %M409.7 : Bool;
   MEJ二级冷凝清洗阀 AT %M410.0 : Bool;
   MSF送风机排水阀 AT %M410.1 : Bool;
   MYF引风机排水阀 AT %M410.2 : Bool;
   MEJ二级冷冻水阀 AT %M410.3 : Bool;
   MQX清洗伸缩气缸 AT %M410.4 : Bool;
   MFK放空比例调节阀 AT %M410.5 : Bool;
   MHF回风加热比例调节阀 AT %M410.6 : Bool;
   MJF进风加热比例调节阀 AT %M410.7 : Bool;
   MYJ一级出料 AT %M411.0 : Bool;
   MEJ二级出料 AT %M411.1 : Bool;
   MBD布袋出料 AT %M411.2 : Bool;
   MSS输送出料 AT %M411.3 : Bool;
   MQG气缸升 AT %M411.4 : Bool;
   MQG气缸降 AT %M411.5 : Bool;
   MYH氧含仪隔断阀 AT %M411.6 : Bool;
   MSN室内排水隔膜泵 AT %M412.0 : Bool;
   MSS输送自整定 AT %M412.1 : Bool;
   MSS输送加热 AT %M412.2 : Bool;
   MBY100 AT %M412.3 : Bool;
   MBY101 AT %M412.4 : Bool;
   MAS室外回水阀 AT %M412.5 : Bool;
   MAS室内回水阀 AT %M412.6 : Bool;
   MSN室内清洗总阀 AT %M412.7 : Bool;
   MHS回水隔断阀1 AT %M413.0 : Bool;
   MAB进水隔断阀 AT %M413.1 : Bool;
   MHSQ回水隔断阀1 AT %M413.2 : Bool;
   MABQ进水隔断阀 AT %M413.3 : Bool;
   MLG料罐清洗阀 AT %M413.4 : Bool;
   MHF回风温度加热 AT %M413.5 : Bool;
   MHF回风加热自整定 AT %M413.6 : Bool;
   MSC四参数控制 AT %M413.7 : Bool;
   MMC脉冲周期_PID AT %M414.0 : Bool;
   MMC脉冲周期_进料 AT %M414.1 : Bool;
   MLS料水手动调节 AT %M414.2 : Bool;
   MXT心跳接受信号 AT %M414.3 : Bool;
   MCS纯水洗请求 AT %M414.4 : Bool;
   MJS碱水洗请求 AT %M414.5 : Bool;
   MRJ溶剂请求 AT %M414.6 : Bool;
   MYG压干请求 AT %M414.7 : Bool;
   MQR确认 AT %M415.0 : Bool;
   MSC四参数手动调节 AT %M415.1 : Bool;
   MZT暂停辅助 AT %M415.2 : Bool;
   MSC四参数开辅助 AT %M415.3 : Bool;
   MSC四参数关辅助 AT %M415.4 : Bool;
   MJL进料调节 AT %M415.5 : Bool;
   MSC四参数调节 AT %M415.6 : Bool;
   MSC四参数手动状态 AT %M415.7 : Bool;
   MJL进料手动状态 AT %M416.1 : Bool;
   MSS输送系统 AT %M416.2 : Bool;
   MJS进水调节 AT %M416.3 : Bool;
   MLS料水系统调节 AT %M416.4 : Bool;
   MKS开始清洗 AT %M416.5 : Bool;
   MJS结束清洗 AT %M416.6 : Bool;
   MZB准备清洗 AT %M416.7 : Bool;
   MCZ初状态 AT %M417.0 : Bool;
   MZD自动清洗 AT %M417.1 : Bool;
   MSD手动_纯水清洗 AT %M417.2 : Bool;
   MSD手动_碱水清洗 AT %M417.3 : Bool;
   MQX清洗辅助 AT %M417.4 : Bool;
   "MSD手动_溶剂清洗(1)" AT %M417.5 : Bool;
   MSD手动_溶剂清洗 AT %M417.6 : Bool;
   MZT主塔伸缩气缸 AT %M417.7 : Bool;
   MZT主塔清洗 AT %M418.0 : Bool;
   MZT总通路 AT %M418.1 : Bool;
   MXY泄压请求 AT %M418.2 : Bool;
   QXY泄压请求 AT %M418.3 : Bool;
   MBJ本机调试模式 AT %M418.4 : Bool;
   MSD手动_二纯水清洗 AT %M418.5 : Bool;
   MFZ仿真调试 AT %M418.6 : Bool;
   MSB设备振打 AT %M418.7 : Bool;
   MQZ前置水阀 AT %M419.0 : Bool;
   MYJ一级旋风振打锤 AT %M419.1 : Bool;
   MEJ二级旋风振打锤 AT %M419.2 : Bool;
   MYJ一级旋风振荡器 AT %M419.3 : Bool;
   MAQ安全停机 AT %M419.4 : Bool;
   MZS注射水请求 AT %M419.5 : Bool;
   MSJ水进程泵 AT %M419.6 : Bool;
   MRJ溶剂进程泵 AT %M419.7 : Bool;
   MGS供水泵 AT %M420.0 : Bool;
   MRC热纯自动洗 AT %M420.1 : Bool;
   MRC热纯加热 AT %M420.2 : Bool;
   MBD本地调试 AT %M420.3 : Bool;
   MRS热水洗请求 AT %M420.4 : Bool;
   MGD管道压力手动调节 AT %M420.5 : Bool;
   MPS排水运行标志 AT %M420.6 : Bool;
END_VAR

VAR_GLOBAL   // PLC tag table "MTX"
   MLS冷水机状态2 AT %MW208 : Int;
   MLS冷水机状态3 AT %MW210 : Int;
   MLS冷水机通信状态 AT %M211.7 : Bool;
   MLS冷水机加热状态 AT %M211.6 : Bool;
   MLS冷水机制冷状态 AT %M211.5 : Bool;
   MLS冷水机超温报警 AT %M209.7 : Bool;
   MLS冷水机低温报警 AT %M209.6 : Bool;
   MLS冷水机压力报警 AT %M209.5 : Bool;
END_VAR

VAR_GLOBAL   // PLC tag table "默认变量表"
   System_Byte AT %MB1 : Byte;
   FirstScan AT %M1.0 : Bool;
   DiagStatusUpdate AT %M1.1 : Bool;
   AlwaysTRUE AT %M1.2 : Bool;
   AlwaysFALSE AT %M1.3 : Bool;
   Clock_Byte AT %MB0 : Byte;
   Clock_10Hz AT %M0.0 : Bool;
   Clock_5Hz AT %M0.1 : Bool;
   "Clock_2.5Hz" AT %M0.2 : Bool;
   Clock_2Hz AT %M0.3 : Bool;
   "Clock_1.25Hz" AT %M0.4 : Bool;
   Clock_1Hz AT %M0.5 : Bool;
   "Clock_0.625Hz" AT %M0.6 : Bool;
   "Clock_0.5Hz" AT %M0.7 : Bool;
   Tag_1 AT %MD800 : Real;
   Tag_2 AT %M810.0 : Bool;
   Tag_3 AT %MD820 : Real;
   Tag_4 AT %MD830 : Real;
   Tag_5 AT %MW840 : Int;
   Tag_6 AT %MD600 : DWord;
   Tag_7 AT %MD610 : DWord;
   Tag_8 AT %MD620 : DWord;
   Tag_9 AT %MD530 : DWord;
   Tag_10 AT %MD840 : DWord;
   Tag_12 AT %M100.0 : Bool;
   Tag_13 AT %M100.1 : Bool;
   自动运行报警 AT %M844.0 : Bool;
   自动停止 AT %M844.1 : Bool;
   Tag_14 AT %M110.0 : Bool;
   Tag_15 AT %M110.1 : Bool;
   Tag_16 AT %M111.0 : Bool;
   Tag_17 AT %M111.1 : Bool;
   M_手动修改 AT %M2000.0 : Bool;
   M_手动设定值 AT %MD2004 : Real;
   Tag_11 AT %MW300 : Word;
   Tag_18 AT %MW320 : Word;
   MQX清洗模式 AT %MW322 : Int;
   QQX清洗模式状态 AT %MW324 : Int;
   TEST AT %M111.2 : Bool;
END_VAR

DATA_BLOCK "485调试"   // DB22
{ S7_Optimized_Access := 'TRUE' }
VERSION : 0.1
// stored: AutoNumber true, DBAccessibleFromOPCUA true, DBAccessibleFromWebserver true, IsOnlyStoredInLoadMemory false, IsRetainMemResEnabled false, IsWriteProtectedInAS false, MemoryReserve 100
   VAR
      done : Bool;
      error : Bool;
      status : Word;
      errorcode : Word;
   END_VAR
BEGIN
END_DATA_BLOCK

DATA_BLOCK "INCIP"   // DB10
{ S7_Optimized_Access := 'TRUE' }
VERSION : 0.1
// stored: AutoNumber true, DBAccessibleFromOPCUA true, DBAccessibleFromWebserver true, IsOnlyStoredInLoadMemory false, IsRetainMemResEnabled false, IsWriteProtectedInAS false, MemoryReserve 100
   VAR
      DD电导合格值 : Real;
      JX碱洗温度设定 : Real := 80.0;
      DD电导率当前值 : Real;
      JX碱洗温度 : Real;
      CIP压力 : Real;
      MZD自动清洗 : Bool;
      MSD手动_纯水清洗 : Bool;
      MSD手动_碱水清洗 : Bool;
      MSD手动_溶剂清洗 : Bool;
      MSD手动_热水清洗 : Bool;
      MQX清洗重置 : Bool;
      MCS纯水罐阀门 : Bool;
      MJS碱水罐阀门 : Bool;
      MZS注射水阀门 : Bool;
      MYK压空吹干阀 : Bool;
      MD清洗失败 : Bool;
      MQX室内清洗辅助 : Bool;
      MZT主塔清洗头 : Bool;
      MZT中途停止 : Bool;
      MXT心跳信号发送 : Bool;
      MXT心跳信号接受 : Bool;
      MXY泄压请求 : Bool;
      MGS供水泵请求 : Bool;
      MCIP远程状态 : Bool;
      QCS纯水罐阀门 : Bool;
      QJS碱水罐阀门 : Bool;
      QZS注射水罐阀门 : Bool;
      QYG压干阀门 : Bool;
      QGS供水泵状态CIP : Bool;
      QXY泄压阀门 : Bool;
      PS排水时间 : Real;
      PS排水时间计时 : Real;
   END_VAR
BEGIN
END_DATA_BLOCK

DATA_BLOCK "INCIPCS"   // DB42
{ S7_Optimized_Access := 'TRUE' }
VERSION : 0.1
// stored: AutoNumber true, DBAccessibleFromOPCUA true, DBAccessibleFromWebserver true, IsOnlyStoredInLoadMemory false, IsRetainMemResEnabled false, IsWriteProtectedInAS false, MemoryReserve 100
   VAR RETAIN
      "1设定时间" : Real := 10.0;
      "2设定时间" : Real := 10.0;
      "3设定时间" : Real := 10.0;
      "4设定时间" : Real := 10.0;
      "5设定时间" : Real := 10.0;
      "6设定时间" : Real := 10.0;
      "7设定时间" : Real := 10.0;
      "8设定时间" : Real := 10.0;
      "9设定时间" : Real := 10.0;
      "10设定时间" : Real := 10.0;
      "11设定时间" : Real := 10.0;
      "12设定时间" : Real := 10.0;
      "13设定时间" : Real := 10.0;
      "14设定时间" : Real := 10.0;
      "15设定时间" : Real := 10.0;
      "16设定时间" : Real := 10.0;
   END_VAR
   VAR
      "0计时" : Real;
      "1计时" : Real;
      "2计时" : Real;
      "3计时" : Real;
      "4计时" : Real;
      "5计时" : Real;
      "6计时" : Real;
      "7计时" : Real;
      "8计时" : Real;
      "9计时" : Real;
      "10计时" : Real;
      "11计时" : Real;
      "12计时" : Real;
      "13计时" : Real;
      "14计时" : Real;
      "15计时" : Real;
      "16计时" : Real;
   END_VAR
BEGIN
END_DATA_BLOCK

DATA_BLOCK "INCIPCS2"   // DB41
{ S7_Optimized_Access := 'TRUE' }
VERSION : 0.1
// stored: AutoNumber true, DBAccessibleFromOPCUA true, DBAccessibleFromWebserver true, IsOnlyStoredInLoadMemory false, IsRetainMemResEnabled false, IsWriteProtectedInAS false, MemoryReserve 100
   VAR RETAIN
      "1设定时间" : Real := 10.0;
      "2设定时间" : Real := 10.0;
      "3设定时间" : Real := 10.0;
      "4设定时间" : Real := 10.0;
      "5设定时间" : Real := 10.0;
      "6设定时间" : Real := 10.0;
      "7设定时间" : Real := 10.0;
      "8设定时间" : Real := 10.0;
      "9设定时间" : Real := 10.0;
      "10设定时间" : Real := 10.0;
      "11设定时间" : Real := 10.0;
      "12设定时间" : Real := 10.0;
      "13设定时间" : Real := 10.0;
      "14设定时间" : Real := 10.0;
      "15设定时间" : Real := 10.0;
      "16设定时间" : Real := 10.0;
   END_VAR
   VAR
      "1计时" : Real;
      "2计时" : Real;
      "3计时" : Real;
      "4计时" : Real;
      "5计时" : Real;
      "6计时" : Real;
      "7计时" : Real;
      "8计时" : Real;
      "9计时" : Real;
      "10计时" : Real;
      "11计时" : Real;
      "12计时" : Real;
      "13计时" : Real;
      "14计时" : Real;
      "15计时" : Real;
      "16计时" : Real;
      "1电导率" : Real;
      "2电导率" : Real;
      "3电导率" : Real;
      "4电导率" : Real;
      "5电导率" : Real;
      "6电导率" : Real;
      "7电导率" : Real;
      "8电导率" : Real;
      "9电导率" : Real;
      "10电导率" : Real;
      "11电导率" : Real;
      "12电导率" : Real;
      "13电导率" : Real;
      "14电导率" : Real;
      "15电导率" : Real;
      "16电导率" : Real;
      "1清洗状态" : Bool;
      "2清洗状态" : Bool;
      "3清洗状态" : Bool;
      "4清洗状态" : Bool;
      "5清洗状态" : Bool;
      "6清洗状态" : Bool;
      "7清洗状态" : Bool;
      "8清洗状态" : Bool;
      "9清洗状态" : Bool;
      "10清洗状态" : Bool;
      "11清洗状态" : Bool;
      "12清洗状态" : Bool;
      "13清洗状态" : Bool;
      "14清洗状态" : Bool;
      "15清洗状态" : Bool;
      "16清洗状态" : Bool;
   END_VAR
BEGIN
END_DATA_BLOCK

DATA_BLOCK "INCIPJS"   // DB40
{ S7_Optimized_Access := 'TRUE' }
VERSION : 0.1
// stored: AutoNumber true, DBAccessibleFromOPCUA true, DBAccessibleFromWebserver true, IsOnlyStoredInLoadMemory false, IsRetainMemResEnabled false, IsWriteProtectedInAS false, MemoryReserve 100
   VAR RETAIN
      "1设定时间" : Real := 10.0;
      "2设定时间" : Real := 10.0;
      "3设定时间" : Real := 10.0;
      "4设定时间" : Real := 10.0;
      "5设定时间" : Real := 10.0;
      "6设定时间" : Real := 10.0;
      "7设定时间" : Real := 10.0;
      "8设定时间" : Real := 10.0;
      "9设定时间" : Real := 10.0;
      "10设定时间" : Real := 10.0;
      "11设定时间" : Real := 10.0;
      "12设定时间" : Real := 10.0;
      "13设定时间" : Real := 10.0;
      "14设定时间" : Real := 10.0;
      "15设定时间" : Real := 10.0;
      "16设定时间" : Real := 10.0;
   END_VAR
   VAR
      "1计时" : Real;
      "2计时" : Real;
      "3计时" : Real;
      "4计时" : Real;
      "5计时" : Real;
      "6计时" : Real;
      "7计时" : Real;
      "8计时" : Real;
      "9计时" : Real;
      "10计时" : Real;
      "11计时" : Real;
      "12计时" : Real;
      "13计时" : Real;
      "14计时" : Real;
      "15计时" : Real;
      "16计时" : Real;
   END_VAR
BEGIN
END_DATA_BLOCK

DATA_BLOCK "INCIPRJ"   // DB15
{ S7_Optimized_Access := 'TRUE' }
VERSION : 0.1
// stored: AutoNumber true, DBAccessibleFromOPCUA true, DBAccessibleFromWebserver true, IsOnlyStoredInLoadMemory false, IsRetainMemResEnabled false, IsWriteProtectedInAS false, MemoryReserve 100
   VAR RETAIN
      "1设定时间" : Real := 10.0;
      "2设定时间" : Real := 10.0;
      "3设定时间" : Real := 10.0;
      "4设定时间" : Real := 10.0;
      "5设定时间" : Real := 10.0;
      "6设定时间" : Real := 10.0;
      "7设定时间" : Real := 10.0;
      "8设定时间" : Real := 10.0;
      "9设定时间" : Real := 10.0;
      "10设定时间" : Real := 10.0;
      "11设定时间" : Real := 10.0;
      "12设定时间" : Real := 10.0;
      "13设定时间" : Real := 10.0;
      "14设定时间" : Real := 10.0;
      "15设定时间" : Real := 10.0;
      "16设定时间" : Real := 10.0;
   END_VAR
   VAR
      "1计时" : Real;
      "2计时" : Real;
      "3计时" : Real;
      "4计时" : Real;
      "5计时" : Real;
      "6计时" : Real;
      "7计时" : Real;
      "8计时" : Real;
      "9计时" : Real;
      "10计时" : Real;
      "11计时" : Real;
      "12计时" : Real;
      "13计时" : Real;
      "14计时" : Real;
      "15计时" : Real;
      "16计时" : Real;
   END_VAR
BEGIN
END_DATA_BLOCK

DATA_BLOCK "INCIPZS"   // DB27
{ S7_Optimized_Access := 'TRUE' }
VERSION : 0.1
// stored: AutoNumber true, DBAccessibleFromOPCUA true, DBAccessibleFromWebserver true, IsOnlyStoredInLoadMemory false, IsRetainMemResEnabled false, IsWriteProtectedInAS false, MemoryReserve 100
   VAR RETAIN
      "1设定时间" : Real := 10.0;
      "2设定时间" : Real := 10.0;
      "3设定时间" : Real := 10.0;
      "4设定时间" : Real := 10.0;
      "5设定时间" : Real := 10.0;
      "6设定时间" : Real := 10.0;
      "7设定时间" : Real := 10.0;
      "8设定时间" : Real := 10.0;
      "9设定时间" : Real := 10.0;
      "10设定时间" : Real := 10.0;
      "11设定时间" : Real := 10.0;
      "12设定时间" : Real := 10.0;
      "13设定时间" : Real := 10.0;
      "14设定时间" : Real := 10.0;
      "15设定时间" : Real := 10.0;
      "16设定时间" : Real := 10.0;
   END_VAR
   VAR
      "1计时" : Real;
      "2计时" : Real;
      "3计时" : Real;
      "4计时" : Real;
      "5计时" : Real;
      "6计时" : Real;
      "7计时" : Real;
      "8计时" : Real;
      "9计时" : Real;
      "10计时" : Real;
      "11计时" : Real;
      "12计时" : Real;
      "13计时" : Real;
      "14计时" : Real;
      "15计时" : Real;
      "16计时" : Real;
   END_VAR
BEGIN
END_DATA_BLOCK

DATA_BLOCK "OUTCIP"   // DB46
{ S7_Optimized_Access := 'TRUE' }
VERSION : 0.1
// stored: AutoNumber true, DBAccessibleFromOPCUA true, DBAccessibleFromWebserver true, IsOnlyStoredInLoadMemory false, IsRetainMemResEnabled false, IsWriteProtectedInAS false, MemoryReserve 100
   VAR
      DD电导合格值 : Real;
      JX碱洗温度设定 : Real := 80.0;
      DD电导率当前值 : Real;
      JX碱洗温度 : Real;
      CIP压力 : Real;
      MZD自动清洗 : Bool;
      MSD手动_纯水清洗 : Bool;
      MSD手动_碱水清洗 : Bool;
      MSD手动_溶剂清洗 : Bool;
      MSD手动_热水清洗 : Bool;
      MQX清洗重置 : Bool;
      MCS纯水罐阀门 : Bool;
      MJS碱水罐阀门 : Bool;
      MZS注射水阀门 : Bool;
      MYK压空吹干阀 : Bool;
      MD清洗失败 : Bool;
      MQX室外清洗辅助 : Bool;
      MZT主塔清洗头 : Bool;
      MZT中途停止 : Bool;
      MXT心跳信号发送 : Bool;
      MXT心跳信号接受 : Bool;
      MXY泄压请求 : Bool;
      MGS供水泵请求 : Bool;
      MCIP远程状态 : Bool;
      QCS纯水罐阀门 : Bool;
      QJS碱水罐阀门 : Bool;
      QZS注射水罐阀门 : Bool;
      QYG压干阀门 : Bool;
      QGS供水泵状态CIP : Bool;
      QXY泄压阀门 : Bool;
      PS排水时间 : Real;
      PS排水时间计时 : Real;
   END_VAR
BEGIN
END_DATA_BLOCK

DATA_BLOCK "OUTCIPCS"   // DB39
{ S7_Optimized_Access := 'TRUE' }
VERSION : 0.1
// stored: AutoNumber true, DBAccessibleFromOPCUA true, DBAccessibleFromWebserver true, IsOnlyStoredInLoadMemory false, IsRetainMemResEnabled false, IsWriteProtectedInAS false, MemoryReserve 100
   VAR RETAIN
      "1设定时间" : Real := 10.0;
      "2设定时间" : Real := 10.0;
      "3设定时间" : Real := 10.0;
      "4设定时间" : Real := 10.0;
      "5设定时间" : Real := 10.0;
      "6设定时间" : Real := 10.0;
      "7设定时间" : Real := 10.0;
      "8设定时间" : Real := 10.0;
      "9设定时间" : Real := 10.0;
      "10设定时间" : Real := 10.0;
      "11设定时间" : Real := 10.0;
      "12设定时间" : Real := 10.0;
      "13设定时间" : Real := 10.0;
      "14设定时间" : Real := 10.0;
      "15设定时间" : Real := 10.0;
      "16设定时间" : Real := 10.0;
   END_VAR
   VAR
      "0计时" : Real;
      "1计时" : Real;
      "2计时" : Real;
      "3计时" : Real;
      "4计时" : Real;
      "5计时" : Real;
      "6计时" : Real;
      "7计时" : Real;
      "8计时" : Real;
      "9计时" : Real;
      "10计时" : Real;
      "11计时" : Real;
      "12计时" : Real;
      "13计时" : Real;
      "14计时" : Real;
      "15计时" : Real;
      "16计时" : Real;
   END_VAR
BEGIN
END_DATA_BLOCK

DATA_BLOCK "OUTCIPCS2"   // DB38
{ S7_Optimized_Access := 'TRUE' }
VERSION : 0.1
// stored: AutoNumber true, DBAccessibleFromOPCUA true, DBAccessibleFromWebserver true, IsOnlyStoredInLoadMemory false, IsRetainMemResEnabled false, IsWriteProtectedInAS false, MemoryReserve 100
   VAR RETAIN
      "1设定时间" : Real := 10.0;
      "2设定时间" : Real := 10.0;
      "3设定时间" : Real := 10.0;
      "4设定时间" : Real := 10.0;
      "5设定时间" : Real := 10.0;
      "6设定时间" : Real := 10.0;
      "7设定时间" : Real := 10.0;
      "8设定时间" : Real := 10.0;
      "9设定时间" : Real := 10.0;
      "10设定时间" : Real := 10.0;
      "11设定时间" : Real := 10.0;
      "12设定时间" : Real := 10.0;
      "13设定时间" : Real := 10.0;
      "14设定时间" : Real := 10.0;
      "15设定时间" : Real := 10.0;
      "16设定时间" : Real := 10.0;
   END_VAR
   VAR
      "1计时" : Real;
      "2计时" : Real;
      "3计时" : Real;
      "4计时" : Real;
      "5计时" : Real;
      "6计时" : Real;
      "7计时" : Real;
      "8计时" : Real;
      "9计时" : Real;
      "10计时" : Real;
      "11计时" : Real;
      "12计时" : Real;
      "13计时" : Real;
      "14计时" : Real;
      "15计时" : Real;
      "16计时" : Real;
      "1电导率" : Real;
      "2电导率" : Real;
      "3电导率" : Real;
      "4电导率" : Real;
      "5电导率" : Real;
      "6电导率" : Real;
      "7电导率" : Real;
      "8电导率" : Real;
      "9电导率" : Real;
      "10电导率" : Real;
      "11电导率" : Real;
      "12电导率" : Real;
      "13电导率" : Real;
      "14电导率" : Real;
      "15电导率" : Real;
      "16电导率" : Real;
      "1清洗状态" : Bool;
      "2清洗状态" : Bool;
      "3清洗状态" : Bool;
      "4清洗状态" : Bool;
      "5清洗状态" : Bool;
      "6清洗状态" : Bool;
      "7清洗状态" : Bool;
      "8清洗状态" : Bool;
      "9清洗状态" : Bool;
      "10清洗状态" : Bool;
      "11清洗状态" : Bool;
      "12清洗状态" : Bool;
      "13清洗状态" : Bool;
      "14清洗状态" : Bool;
      "15清洗状态" : Bool;
      "16清洗状态" : Bool;
   END_VAR
BEGIN
END_DATA_BLOCK

DATA_BLOCK "OUTCIPJS"   // DB37
{ S7_Optimized_Access := 'TRUE' }
VERSION : 0.1
// stored: AutoNumber true, DBAccessibleFromOPCUA true, DBAccessibleFromWebserver true, IsOnlyStoredInLoadMemory false, IsRetainMemResEnabled false, IsWriteProtectedInAS false, MemoryReserve 100
   VAR RETAIN
      "1设定时间" : Real := 10.0;
      "2设定时间" : Real := 10.0;
      "3设定时间" : Real := 10.0;
      "4设定时间" : Real := 10.0;
      "5设定时间" : Real := 10.0;
      "6设定时间" : Real := 10.0;
      "7设定时间" : Real := 10.0;
      "8设定时间" : Real := 10.0;
      "9设定时间" : Real := 10.0;
      "10设定时间" : Real := 10.0;
      "11设定时间" : Real := 10.0;
      "12设定时间" : Real := 10.0;
      "13设定时间" : Real := 10.0;
      "14设定时间" : Real := 10.0;
      "15设定时间" : Real := 10.0;
      "16设定时间" : Real := 10.0;
   END_VAR
   VAR
      "1计时" : Real;
      "2计时" : Real;
      "3计时" : Real;
      "4计时" : Real;
      "5计时" : Real;
      "6计时" : Real;
      "7计时" : Real;
      "8计时" : Real;
      "9计时" : Real;
      "10计时" : Real;
      "11计时" : Real;
      "12计时" : Real;
      "13计时" : Real;
      "14计时" : Real;
      "15计时" : Real;
      "16计时" : Real;
   END_VAR
BEGIN
END_DATA_BLOCK

DATA_BLOCK "OUTCIPRJ"   // DB7
{ S7_Optimized_Access := 'TRUE' }
VERSION : 0.1
// stored: AutoNumber true, DBAccessibleFromOPCUA true, DBAccessibleFromWebserver true, IsOnlyStoredInLoadMemory false, IsRetainMemResEnabled false, IsWriteProtectedInAS false, MemoryReserve 100
   VAR RETAIN
      "1设定时间" : Real := 10.0;
      "2设定时间" : Real := 10.0;
      "3设定时间" : Real := 10.0;
      "4设定时间" : Real := 10.0;
      "5设定时间" : Real := 10.0;
      "6设定时间" : Real := 10.0;
      "7设定时间" : Real := 10.0;
      "8设定时间" : Real := 10.0;
      "9设定时间" : Real := 10.0;
      "10设定时间" : Real := 10.0;
      "11设定时间" : Real := 10.0;
      "12设定时间" : Real := 10.0;
      "13设定时间" : Real := 10.0;
      "14设定时间" : Real := 10.0;
      "15设定时间" : Real := 10.0;
      "16设定时间" : Real := 10.0;
   END_VAR
   VAR
      "1计时" : Real;
      "2计时" : Real;
      "3计时" : Real;
      "4计时" : Real;
      "5计时" : Real;
      "6计时" : Real;
      "7计时" : Real;
      "8计时" : Real;
      "9计时" : Real;
      "10计时" : Real;
      "11计时" : Real;
      "12计时" : Real;
      "13计时" : Real;
      "14计时" : Real;
      "15计时" : Real;
      "16计时" : Real;
   END_VAR
BEGIN
END_DATA_BLOCK

DATA_BLOCK "OUTCIPZS"   // DB47
{ S7_Optimized_Access := 'TRUE' }
VERSION : 0.1
// stored: AutoNumber true, DBAccessibleFromOPCUA true, DBAccessibleFromWebserver true, IsOnlyStoredInLoadMemory false, IsRetainMemResEnabled false, IsWriteProtectedInAS false, MemoryReserve 100
   VAR RETAIN
      "1设定时间" : Real := 10.0;
      "2设定时间" : Real := 10.0;
      "3设定时间" : Real := 10.0;
      "4设定时间" : Real := 10.0;
      "5设定时间" : Real := 10.0;
      "6设定时间" : Real := 10.0;
      "7设定时间" : Real := 10.0;
      "8设定时间" : Real := 10.0;
      "9设定时间" : Real := 10.0;
      "10设定时间" : Real := 10.0;
      "11设定时间" : Real := 10.0;
      "12设定时间" : Real := 10.0;
      "13设定时间" : Real := 10.0;
      "14设定时间" : Real := 10.0;
      "15设定时间" : Real := 10.0;
      "16设定时间" : Real := 10.0;
   END_VAR
   VAR
      "1计时" : Real;
      "2计时" : Real;
      "3计时" : Real;
      "4计时" : Real;
      "5计时" : Real;
      "6计时" : Real;
      "7计时" : Real;
      "8计时" : Real;
      "9计时" : Real;
      "10计时" : Real;
      "11计时" : Real;
      "12计时" : Real;
      "13计时" : Real;
      "14计时" : Real;
      "15计时" : Real;
      "16计时" : Real;
   END_VAR
BEGIN
END_DATA_BLOCK

DATA_BLOCK "BDBS"   // DB45
{ S7_Optimized_Access := 'TRUE' }
VERSION : 0.1
// stored: AutoNumber true, DBAccessibleFromOPCUA true, DBAccessibleFromWebserver true, IsOnlyStoredInLoadMemory false, IsRetainMemResEnabled false, IsWriteProtectedInAS false, MemoryReserve 100
   VAR
      SJ事件记录_ { ExternalWritable := 'False'} : Array[1..20] of String[20];
      SJ事件编号 { ExternalWritable := 'False'} : Array[1..20] of Int;
      QL清零 : Bool;
   END_VAR
BEGIN
END_DATA_BLOCK

DATA_BLOCK "BDKS"   // DB43
{ S7_Optimized_Access := 'TRUE' }
VERSION : 0.1
// stored: AutoNumber true, DBAccessibleFromOPCUA true, DBAccessibleFromWebserver true, IsOnlyStoredInLoadMemory false, IsRetainMemResEnabled false, IsWriteProtectedInAS false, MemoryReserve 100
   VAR
      SJ事件记录_ { ExternalWritable := 'False'} : Array[1..20] of String[20];
      SJ事件编号 { ExternalWritable := 'False'} : Array[1..20] of Int;
      QL清零 : Bool;
   END_VAR
BEGIN
END_DATA_BLOCK

DATA_BLOCK "BS"   // DB44
{ S7_Optimized_Access := 'TRUE' }
VERSION : 0.1
// stored: AutoNumber true, DBAccessibleFromOPCUA true, DBAccessibleFromWebserver true, IsOnlyStoredInLoadMemory false, IsRetainMemResEnabled false, IsWriteProtectedInAS false, MemoryReserve 100
   VAR RETAIN
      JF进风流量上阈值 : Real := 150.0;
      JF进风流量下阈值 : Real := 150.0;
      ZT主塔压力引风升临界 : Real := 900.0;
      JF进风流量引风关临界 : Real := 2000.0;
      JF进风流量送风关临界 : Real := 1300.0;
      SF送风机1分钟升速 : Real := 4.0;
      YP预喷雾检测主塔压力维持时间 : Int := 30;
      YP预喷雾检测高压 : Real := 800.0;
      YP预喷雾检测低压 : Real := -300.0;
      YP预喷雾检测系统结果 : Int := 1;
      YP预喷雾检测系统正常 : Bool := TRUE;
      YP预喷雾进风流量 : Real := 1500.0;
      "YP预喷雾-离雾-进温" : Real := 100.0;
      "YP预喷雾-离雾-出温" : Real := 85.0;
      YP预喷雾温稳正式时间 : Int := 100;
      GJ关机洗喷头时间 : Int := 60;
      "GJ关机-停水-出温" : Real := 110.0;
      "GJ关机-停水-停雾" : DInt := 60;
      "GJ关机-四参数关-进温" : Real := 70.0;
      "GJ关机-输送-送温" : Real := 65.0;
      ZD自动运行报警 : Bool := FALSE;
      BD步段运行_秒 : Int := 0;
      BD步段运行_分 : Int := 0;
      BD步段运行_时 : Int := 0;
      ZY总运行_秒 : Int := 0;
      ZY总运行_分 : Int := 0;
      ZY总运行_时 : Int := 0;
      JL进料_时 : Int := 0;
      JL进料_分 : Int := 0;
      JL进料_秒 : Int := 0;
      BD步段设定 : Int := 0;
      BD步段运行 : Int := 0;
      ZD自动停止 : Bool := FALSE;
      AQ安全停机 : Bool := FALSE;
      JL进料时间设定 : Real := 10.0;
      XT系统状态 : Int := 1;
      JL进料进风阈值 : Real := 5.0;
      JL进料出风条件 : Real := 80.0;
   END_VAR
   VAR
      WQ尾气温度设定 : Real := 30.0;
      CF出温高报 : Real := 110.0;
      CF出温高高报 : Real := 130.0;
      WQ尾温高报 : Real := 35.0;
      WQ尾温高高报 : Real := 40.0;
      JF进温高报 : Real := 130.0;
      JF进温高高报 : Real := 150.0;
   END_VAR
BEGIN
END_DATA_BLOCK

DATA_BLOCK "BY1"   // DB9
{ S7_Optimized_Access := 'TRUE' }
VERSION : 0.1
// stored: AutoNumber true, DBAccessibleFromOPCUA true, DBAccessibleFromWebserver true, IsOnlyStoredInLoadMemory false, IsRetainMemResEnabled false, IsWriteProtectedInAS false, MemoryReserve 100
   VAR
      MBY等待保压 : Bool := FALSE;
      MBY正在充气 : Bool := TRUE;
      MBY保压不佳 : Bool := FALSE;
      MBY正在保压 : Bool := FALSE;
      MBY保压正常 : Bool := FALSE;
      MBY保压 : Bool := TRUE;
      MQT其他阀 : Bool := FALSE;
      MCQ充气阀 : Bool := FALSE;
      当前阶段 : Int := 1;
   END_VAR
   VAR RETAIN
      SV低设定 : Real := 1000.0;
      SV高设定 : Real := 3000.0;
      SV保压差值 : Real := 1000.0;
      SV保压时 : UInt := 0;
      SV保压分 : UInt := 0;
      SV保压秒 : UInt := 30;
   END_VAR
   VAR
      PV塔内压力 : Real := 0.0;
      PV保压前 : Real := 1016.367;
      PV保压后 : Real := 1016.367;
      PV当前差值 : Real := 0.0;
      PV保压时 : UInt := 0;
      PV保压分 : UInt := 0;
      PV保压秒 : UInt := 30;
      BY保压重置 : Bool := FALSE;
   END_VAR
BEGIN
END_DATA_BLOCK

DATA_BLOCK "BY2"   // DB24
{ S7_Optimized_Access := 'TRUE' }
VERSION : 0.1
// stored: AutoNumber true, DBAccessibleFromOPCUA true, DBAccessibleFromWebserver true, IsOnlyStoredInLoadMemory false, IsRetainMemResEnabled false, IsWriteProtectedInAS false, MemoryReserve 100
   VAR
      MBY等待保压 : Bool;
      MBY正在充气 : Bool;
      MBY保压不佳 : Bool;
      MBY正在保压 : Bool;
      MBY保压正常 : Bool;
      MBY保压 : Bool;
      MQT其他阀 : Bool;
      MCQ充气阀 : Bool;
      当前阶段 : Int;
   END_VAR
   VAR RETAIN
      SV低设定 : Real;
      SV高设定 : Real;
      SV保压差值 : Real;
      SV保压时 : UInt;
      SV保压分 : UInt;
      SV保压秒 : UInt;
   END_VAR
   VAR
      PV塔内压力 : Real;
      PV保压前 : Real;
      PV保压后 : Real;
      PV当前差值 : Real;
      PV保压时 : UInt;
      PV保压分 : UInt;
      PV保压秒 : UInt;
   END_VAR
BEGIN
END_DATA_BLOCK

DATA_BLOCK "CIP_CUS"   // DB6
{ S7_Optimized_Access := 'FALSE' }
VERSION : 0.1
// stored: AutoNumber true, DBAccessibleFromOPCUA true, DBAccessibleFromWebserver true, IsOnlyStoredInLoadMemory false, IsWriteProtectedInAS false
   VAR
      RCV : Struct
         QXT心跳信号 : Bool;
         QCIP启动 : Bool;
         QCS纯水洗 : Bool;
         QJS碱水洗 : Bool;
         QRJ溶剂洗 : Bool;
         QYK压空阀 : Bool;
         QRS热水洗 : Bool;
         QSJ水进程泵 : Bool;
         QRJ溶剂进程泵 : Bool;
         QXY泄压请求 : Bool;
         QQS缺水状态 : Bool;
         QQX清洗模式状态 : Int;
         QJX碱洗温度 : Real;
         QJS碱水液位 : Real;
         QCS纯水温度 : Real;
         QCS纯水液位 : Real;
         QRJ溶剂温度 : Real;
         QRJ溶剂液位 : Real;
         QJC碱纯压力 : Real;
         QCS溶剂压力 : Real;
      END_STRUCT;
      Send : Struct
         MXT心跳信号 : Bool;
         MBM北面喷雾 : Bool;
         MCS纯水模块洗 : Bool;
         MJS碱水模块洗 : Bool;
         MRJ溶剂模块洗 : Bool;
         MRS热水模块洗 : Bool;
         MCS纯水洗 : Bool;
         MJX碱洗 : Bool;
         MRJ溶剂洗 : Bool;
         MYK压空阀 : Bool;
         MRS热水洗 : Bool;
         MSJ水进程泵 : Bool;
         MRJ溶剂进程泵 : Bool;
         MGS供水泵 : Bool;
         MXY泄压阀 : Bool;
         MQX清洗模式 : Int;
         MPW喷雾模式 : Real;
         MJX碱洗温度设定 : Real := 80.0;
         MPS排水时间 : Real;
      END_STRUCT;
   END_VAR
BEGIN
END_DATA_BLOCK

DATA_BLOCK "DH"   // DB19
{ S7_Optimized_Access := 'TRUE' }
VERSION : 0.1
// stored: AutoNumber true, DBAccessibleFromOPCUA true, DBAccessibleFromWebserver true, IsOnlyStoredInLoadMemory false, IsRetainMemResEnabled false, IsWriteProtectedInAS false, MemoryReserve 100
   VAR
      XH循环风机动画 : Int;
      JL进料泵动画 : Int;
      JB搅拌电机动画 : Int;
      主管道动画 : Int;
      YF引风机动画 : Int;
      SF送风机动画 : Int;
      LX离心雾化动画 : Int;
   END_VAR
BEGIN
END_DATA_BLOCK

DATA_BLOCK "KS"   // DB16
{ S7_Optimized_Access := 'TRUE' }
VERSION : 0.1
// stored: AutoNumber true, DBAccessibleFromOPCUA true, DBAccessibleFromWebserver true, IsOnlyStoredInLoadMemory false, IsRetainMemResEnabled false, IsWriteProtectedInAS false, MemoryReserve 100
   VAR RETAIN
      JF进风流量上阈值 : Real := 150.0;
      JF进风流量下阈值 : Real := 150.0;
      ZT主塔压力引风升临界 : Real := 900.0;
      JF进风流量引风关临界 : Real := 2000.0;
      JF进风流量送风关临界 : Real := 1300.0;
      SF送风机1分钟升速 : Real := 4.0;
      YP预喷雾检测主塔压力维持时间 : Int := 30;
      YP预喷雾检测高压 : Real := 800.0;
      YP预喷雾检测低压 : Real := -300.0;
      YP预喷雾检测系统结果 : Int := 1;
      YP预喷雾检测系统正常 : Bool := TRUE;
      YP预喷雾进风流量 : Real := 2000.0;
      "YP预喷雾-离雾-进温" : Real := 145.0;
      "YP预喷雾-离雾-出温" : Real := 100.0;
      YP预喷雾温稳正式时间 : Int := 90;
      GJ关机洗喷头时间 : Int := 200;
      "GJ关机-停水-出温" : Real := 110.0;
      "GJ关机-停水-停雾" : DInt := 120;
      "GJ关机-四参数关-进温" : Real := 80.0;
      "GJ关机-输送-送温" : Real := 65.0;
      ZD自动运行报警 : Bool := FALSE;
      BD步段运行_秒 : Int := 0;
      BD步段运行_分 : Int := 0;
      BD步段运行_时 : Int := 0;
      ZY总运行_秒 : Int := 0;
      ZY总运行_分 : Int := 0;
      ZY总运行_时 : Int := 0;
      JL进料_时 : Int := 0;
      JL进料_分 : Int := 0;
      JL进料_秒 : Int := 0;
      BD步段设定 : Int := 0;
      BD步段运行 : Int := 0;
      ZD自动停止 : Bool := FALSE;
      AQ安全停机 : Bool := FALSE;
      JL进料时间设定 : Real := 10.0;
      XT系统状态 : Int := 1;
      JL进料进风阈值 : Real := 5.0;
      JL进料出风条件 : Real := 115.0;
   END_VAR
   VAR
      CF出温高报 : Real := 150.0;
      CF出温高高报 : Real := 200.0;
      WQ尾温高报 : Real := 35.0;
      WQ尾温高高报 : Real := 40.0;
      JF进温高报 : Real := 220.0;
      JF进温高高报 : Real := 250.0;
   END_VAR
BEGIN
END_DATA_BLOCK

DATA_BLOCK "PW"   // DB12
{ S7_Optimized_Access := 'FALSE' }
VERSION : 0.1
// stored: AutoNumber true, DBAccessibleFromOPCUA true, DBAccessibleFromWebserver true, IsOnlyStoredInLoadMemory false, IsWriteProtectedInAS false
   VAR RETAIN
      PH批号输入 : Int;
      MS模式设定 : Real;
      AQ安全停机 : Bool;
      自动运行报警 : Bool;
      自动停止 : Bool;
      MS模式状态 : Int;
      ZT总通路 : Int;
   END_VAR
BEGIN
END_DATA_BLOCK

DATA_BLOCK "SD"   // DB21
{ S7_Optimized_Access := 'TRUE' }
VERSION : 0.1
// stored: AutoNumber true, DBAccessibleFromOPCUA true, DBAccessibleFromWebserver true, IsOnlyStoredInLoadMemory false, IsRetainMemResEnabled false, IsWriteProtectedInAS false, MemoryReserve 100
   VAR
      KS开始喷雾 : Bool;
      JS结束喷雾 : Bool;
      FW复位 : Bool;
      XT系统状态 : String;
      XT系统检测结果 : String;
      XT系统正常 : Bool;
      PW喷雾开始标志 : Bool;
      PW喷雾结束标志 : Bool;
      CL处理物料总量 : Real;
      YX运行时间显示 : String;
   END_VAR
BEGIN
END_DATA_BLOCK

DATA_BLOCK "SV"   // DB14
{ S7_Optimized_Access := 'FALSE' }
VERSION : 0.1
// stored: AutoNumber true, DBAccessibleFromOPCUA true, DBAccessibleFromWebserver true, IsOnlyStoredInLoadMemory false, IsWriteProtectedInAS false
   VAR RETAIN
      BD布袋压差高报 : Real := 3000.0;
      BD布袋压差高高报 : Real := 3800.0;
      JF进风压差高报 : Real := 3000.0;
      JF进风压差高高报 : Real := 3800.0;
      TN塔内压力高高报 : Real := 14000.0;
      GD管道压力高报 : Real := 1500.0;
      GD管道压力高高报 : Real := 3000.0;
      GD管道压力设定 : Real := 700.0;
      TN塔内压力低报 : Real := -1000.0;
      TN塔内压力低低报 : Real := -1500.0;
      XH循风机频率设定 : Real := 35.0;
      YF引风频率设定 : Real := 30.0;
      JL进料泵频率设定 : Real := 11.0;
      JF进风温度设定 : Real := 110.0;
      CF出温异常设定 : Real := 0.0;
      JF进温高报 : Real := 220.0;
      JF进温高高报 : Real := 250.0;
      CF出风温度设定 : Real := 30.0;
      CF出温高报 : Real := 150.0;
      CF出温高高报 : Real := 200.0;
      WQ尾温高报 : Real := 35.0;
      WQ尾温高高报 : Real := 40.0;
      BD布袋反吹时间 : Real := 5.0;
      TW塔外气锤时间 : Real := 2.0;
      TN塔内气扫时间 : Real := 2.0;
      DQ氮气下限设定 : Real := 0.0;
      TN塔内压力高报 : Real := 11000.0;
      JW降温温度设定 : Real := 0.0;
      LS冷水温度写 : Real := 0.0;
      ZT主塔振打间隔 : Real := 0.0;
      TZ通针时间 : Real := 0.0;
      PM屏幕编号 : Real := 5.0;
      YH氧含仪高报 : Real := 5.0;
      JD进氮压力 : Real := 0.0;
      JL进料压力高报 : Real := 1500.0;
      JL进料压力高高报 : Real := 2000.0;
      WQ尾气温度 : Real := 35.0;
      JF进风保护温度 : Real := 50.0;
      YH氧含差值 : Real := 10.0;
      YH氧含仪1 : Real := 3.0;
      YH氧含仪2 : Real := 0.0;
      LS冷水检测写 : Real := 0.0;
      JF进风检测写 : Real := 0.0;
      QT气体检测仪低报 : Real := 0.0;
      QT气体检测仪低低报 : Real := 0.0;
      LX离心雾化 : Real := 42.0;
      DQ氮气加热写 : Real := 0.0;
      BD布袋振打时间 : Real := 0.0;
      PS排水延长时间 : Real := 0.0;
      AQ安全比例阀 : Real := 0.0;
      PK排空比例阀 : Real := 0.0;
      JB搅拌电机 : Real := 0.0;
      JF进风加热比例调节阀 : Real := 0.0;
      HF回风加热比例调节阀 : Real := 0.0;
      FK放空比例调节阀 : Real := 0.0;
      SF送风频率 : Real := 25.0;
      SS输送温度设定 : Real := 60.0;
      BD布袋出料设定 : Real := 0.0;
      YJ一级旋风出料设定 : Real := 0.0;
      EJ二级旋风出料设定 : Real := 0.0;
      BD布袋T出料设定 : Real := 0.0;
      YJ一级旋风T出料设定 : Real := 0.0;
      EJ二级旋风T出料设定 : Real := 0.0;
      BD布袋上阀开时间 : Real := 500.0;
      BD布袋上阀关时间 : Real := 3.0;
      BD布袋下阀开时间 : Real := 30.0;
      BD布袋下阀关时间 : Real := 3.0;
      YJ一级旋风上阀开时间 : Real := 300.0;
      YJ一级旋风上阀关时间 : Real := 3.0;
      YJ一级旋风下阀开时间 : Real := 30.0;
      YJ一级旋风下阀关时间 : Real := 3.0;
      EJ二级旋风上阀开时间 : Real := 400.0;
      EJ二级旋风上阀关时间 : Real := 3.0;
      EJ二级旋风下阀开时间 : Real := 30.0;
      EJ二级旋风下阀关时间 : Real := 3.0;
      HF回风温度设定 : Real := 0.0;
      ZT主塔压力设定 : Real := -200.0;
      KQ空气流量设定 : Real := 0.0;
      JL进料流量设定 : Real := 0.0;
      JL进料泵频率手动设定 : Real := 11.0;
      YF引风频率手动设定 : Real := 30.0;
      JF进风流量设定 : Real := 2400.0;
      YF引风频率自动设定 : Real := 30.0;
      JL进料频率自动设定 : Real := 11.0;
      FD阀导气压低报 : Real := 1.0;
      FD阀导气压低低报 : Real := 1.0;
      JF进风压差低报 : Real := 0.0;
      WH雾化油压低报 : Real := -1.0;
      WH雾化油压低低报 : Real := -1.0;
      JD进氮压力低报 : Real := 0.0;
      JD进氮压力低低报 : Real := 0.0;
      CF出风高效高报 : Real := 3000.0;
      CF出风高效高高报 : Real := 3800.0;
      CF出风高效低报 : Real := -50.0;
      SF输送高效高报 : Real := 0.0;
      SF输送高效高高报 : Real := 0.0;
      SF输送高效低报 : Real := 0.0;
      HF回风温度高报 : Real := 80.0;
      HF回风温度高高报 : Real := 100.0;
      BD布袋压差低报 : Real := -50.0;
      SS输送保护温度 : Real := 0.0;
      JL进料停机阈值 : Real := 30.0;
      SB设备振打间隔 : Real := 0.0;
      SS输送温度高高报 : Real := 110.0;
      SS输送温度高报 : Real := 102.0;
      SS输送压差高高报 : Real := 3800.0;
      SS输送压差高报 : Real := 3000.0;
      SS输送压差低报 : Real := -50.0;
      YJ一级液位高报 : Real := 400.0;
      YJ一级液位计高高报 : Real := 500.0;
      EJ二级液位计高报 : Real := 400.0;
      EJ二级液位计高高报 : Real := 500.0;
      CW除雾液位计高报 : Real := 400.0;
      CW除雾液位计高高报 : Real := 500.0;
      FD阀岛气压低报 : Real := 0.0;
      FD阀岛气压低低报 : Real := 0.0;
      YH氧含仪高高报 : Real := 12.0;
      JF进风流量低低报 : Real := 0.0;
      JF进风流量低报 : Real := 0.0;
      QZ前置水罐液位低报 : Real := 150.0;
      QZ前置水罐液位低低报 : Real := 100.0;
      JL进料流量低报 : Real := 0.0;
      JL进料流量低低报 : Real := 0.0;
      YJ一级旋风振打间隔 : Real := 6.0;
      EJ二级旋风振打间隔 : Real := 6.0;
      YJ一级旋风振荡运行 : Real := 3.0;
      YJ一级旋风振荡停止 : Real := 3.0;
      TJ调节单元 : Real := 4.0;
      TJ调节时间 : Real := 60.0;
      BD布袋压差自动反吹 : Real := 3500.0;
      BD布袋压差自动反吹时间 : Real := 1600.0;
      "ZT 中途停止温度分界" : Real := 115.0;
      JX碱洗温度设定 : Real := 0.0;
      FK放空阀手动设定 : Real := 0.0;
      FK放空阀自动设定 : Real := 0.0;
   END_VAR
BEGIN
END_DATA_BLOCK

DATA_BLOCK "YB"   // DB26
{ S7_Optimized_Access := 'TRUE' }
VERSION : 0.1
// stored: AutoNumber true, DBAccessibleFromOPCUA true, DBAccessibleFromWebserver true, IsOnlyStoredInLoadMemory false, IsRetainMemResEnabled false, IsWriteProtectedInAS false, MemoryReserve 100
   VAR
      读重量 : Real;
      A瞬时流量 : Real;
      A瞬时流速 : Real;
      A介质温度 : Real;
      A当前采集 : Real;
      A当前电流 : Real;
      A流速下限 : Real;
      A流速上限 : Real;
      A管道内径 : Real;
      B瞬时流量 : Real;
      B瞬时流速 : Real;
      B介质温度 : Real;
      B当前采集 : Real;
      B当前电流 : Real;
      B流速下限 : Real;
      B流速上限 : Real;
      B管道内径 : Real;
      秤状态 : Array[0..15] of Bool;
      秤操作 : Array[0..2] of Bool;
   END_VAR
BEGIN
END_DATA_BLOCK

ORGANIZATION_BLOCK "Main"   // OB1, SCL, ProgramCycle
TITLE = "Main Program Sweep (Cycle)"
{ S7_Optimized_Access := 'TRUE' }
VERSION : 0.1
// stored: AutoNumber true, IsIECCheckEnabled false, SetENOAutomatically false
   VAR_INPUT
      Initial_Call : Bool;   // Initial call of this OB
      Remanence : Bool;   // =True, if remanent data are available
   END_VAR
BEGIN
   "0- IO Configure"();
   "A1-阀带反馈_DB"();
   "A2-阀带阀导_DB"();
   "A3-电机控制_DB"();
   "A4-脉冲控制_DB"();
   "A6-模拟量输入_DB"();
   "A5-模拟量输出_DB"();
   "A7-温度控制_DB"();
   "6-ALLALARM_DB"();
   "B2--局部连锁_DB"();
   "B3-全局连锁_DB"();
   "B4-清洗连锁_DB"();
   "C1-开式自动_DB"();
   "C2-闭式自动_DB"();
   "C3-室内CIP清洗_DB"();
   "C4-室外CIP清洗_DB"();
   "D1-室内CIP通讯_DB"();
   "D2-室外CIP通讯_DB"();
END_ORGANIZATION_BLOCK

FUNCTION_BLOCK "A1-阀带反馈"   // FB18, SCL
{ S7_Optimized_Access := 'TRUE' }
VERSION : 0.1
// stored: AutoNumber true, IsIECCheckEnabled false, IsRetainMemResEnabled false, MemoryReserve 100, SetENOAutomatically false, UDAEnableTagReadback false
   VAR
      泄压阀 { S7_SetPoint := 'True'} : "A3-普通阀控制";
      进风冷却水阀 { S7_SetPoint := 'True'} : "A3-普通阀控制";
      输送进风阀 { S7_SetPoint := 'True'} : "A3-普通阀控制";
      气流雾化阀 { S7_SetPoint := 'True'} : "A3-普通阀控制";
      开式排风隔断阀 { S7_SetPoint := 'True'} : "A3-普通阀控制";
      闭式排风隔断阀 { S7_SetPoint := 'True'} : "A3-普通阀控制";
      开式进风隔断阀 { S7_SetPoint := 'True'} : "A3-普通阀控制";
      闭式进风隔断阀 { S7_SetPoint := 'True'} : "A3-普通阀控制";
      一级冷却水阀 { S7_SetPoint := 'True'} : "A3-普通阀控制";
      二级冷冻水阀 { S7_SetPoint := 'True'} : "A3-普通阀控制";
      一级排液阀 { S7_SetPoint := 'True'} : "A3-普通阀控制";
      二级排液阀 { S7_SetPoint := 'True'} : "A3-普通阀控制";
      除雾排液阀 { S7_SetPoint := 'True'} : "A3-普通阀控制";
      补氮阀 : "A3-普通阀控制";
      进氮阀 { S7_SetPoint := 'True'} : "A3-普通阀控制";
      塔顶清洗球阀 { S7_SetPoint := 'True'} : "A3-普通阀控制";
      溶剂回收排放阀 { S7_SetPoint := 'True'} : "A3-普通阀控制";
      室内排水隔膜泵 { S7_SetPoint := 'True'} : "A3-普通阀控制";
      溶剂排液泵 { S7_SetPoint := 'True'} : "A3-普通阀控制";
      清洗伸缩气缸 { S7_SetPoint := 'True'} : "A3-普通阀控制";
   END_VAR
BEGIN
   REGION 带反馈控制阀
      // "ALQ冷却水流量低报警"



       IF "MJF进风加热比例调节阀" THEN
           "QJF进风蒸汽比例调节阀" := 1;
       ELSE
           "QJF进风蒸汽比例调节阀" := 0;
       END_IF;

       IF "MJF进风蒸汽开关阀" THEN
           "QJF进风蒸汽开关阀" := 1;
       ELSE
           "QJF进风蒸汽开关阀" := 0;
       END_IF;

       IF "MJF进风蒸汽排水阀" THEN
           "QJF进风蒸汽排水阀" := 1;
       ELSE
           "QJF进风蒸汽排水阀" := 0;
       END_IF;

       IF "MHF回风蒸汽排水阀" THEN
           "QHF回风蒸汽排水阀" := 1;
       ELSE
           "QHF回风蒸汽排水阀" :=0;
       END_IF;



           IF "MSF输送风机" THEN
               "QSS输送风机" := 1;
           ELSE
               "QSS输送风机" := 0;
           END_IF;


           IF "MRJ溶剂排液泵" THEN
               "QRJ溶剂排液泵" := 1;
           ELSE
               "QRJ溶剂排液泵" := 0;
           END_IF;


           IF "MSN室内排水隔膜泵" THEN
               "QSN室内排水隔膜泵" := 1;
           ELSE
               "QSN室内排水隔膜泵" := 0;
           END_IF;


           IF "MCC除尘脉冲" THEN
               "QCC除尘脉冲" := 1;
           ELSE
               "QCC除尘脉冲" := 0;
           END_IF;



           #泄压阀(模式设定 := "PW".MS模式设定,
                条件1 := 0.0,
                条件2 := 0.0,
                阀开信号 := "IXY泄压阀开反馈",
                阀关信号 := "IXY泄压阀关反馈",
                手动控制按钮开 := "MXY泄压阀",
                阀状态 := "QXY泄压阀",
                阀开报警 := "AXY泄压阀开报警",
                阀关报警 := "AXY泄压阀关报警");

           #进风冷却水阀(模式设定 := "PW".MS模式设定,
                   条件1 := 0.0,
                   条件2 := 0.0,
                   阀开信号 := "IJF进风冷却水阀开反馈",
                   阀关信号 := "IJF进风冷却水阀关反馈",
                   手动控制按钮开 := "MJF进风冷却水阀",
                   阀状态 := "QJF进风冷却水阀",
                   阀开报警 := "AJF进风冷却水阀开报警",
                   阀关报警 := "AJF进风冷却水阀关报警");

           #输送进风阀(模式设定 := "PW".MS模式设定,
                  条件1 := 0.0,
                  条件2 := 0.0,
                  阀开信号 := "ISF输送进风阀开反馈",
                  阀关信号 := "ISF输送进风阀关反馈",
                  手动控制按钮开 := "MSS输送进风阀",
                  阀状态 := "QSS输送进风阀",
                  阀开报警 := "ASS输送进风阀开报警",
                  阀关报警 := "ASS输送进风阀关报警");

           #气流雾化阀(模式设定 := "PW".MS模式设定,
                  条件1 := 0.0,
                  条件2 := 0.0,
                  阀开信号 := "IQL气流雾化阀开反馈",
                  阀关信号 := "IQL气流雾化阀关反馈",
                  手动控制按钮开 := "MQL气流雾化阀",
                  阀状态 := "QQL气流雾化阀",
                  阀开报警 := "AQL气流雾化阀开报警",
                  阀关报警 := "AQL气流雾化阀关报警");


           #开式排风隔断阀(模式设定 := "PW".MS模式设定,
                    条件1 := 0.0,
                    条件2 := 0.0,
                    阀开信号 := "IKS开式排风隔断阀开反馈",
                    阀关信号 := "IKS开式排风隔断阀关反馈",
                    手动控制按钮开 := "MKS开式排风隔断阀",
                    阀状态 := "QKS开式排风隔断阀",
                    阀开报警 := "AKS开式排风隔断阀开报警",
                    阀关报警 := "AKS开式排风隔断阀关报警");

           #闭式排风隔断阀(模式设定 := "PW".MS模式设定,
                    条件1 := 0.0,
                    条件2 := 0.0,
                    阀开信号 := "IBS闭式排风隔断阀开反馈",
                    阀关信号 := "IBS闭式排风隔断阀关反馈",
                    手动控制按钮开 := "MBS闭式排风隔断阀",
                    阀状态 := "QBS闭式排风隔断阀",
                    阀开报警 := "ABS闭式排风隔断阀开报警",
                    阀关报警 := "ABS闭式排风隔断阀关报警");

           #开式进风隔断阀(模式设定 := "PW".MS模式设定,
                    条件1 := 0.0,
                    条件2 := 0.0,
                    阀开信号 := "IKS开式进风隔断阀开反馈",
                    阀关信号 := "IKS开式进风隔断阀关反馈",
                    手动控制按钮开 := "MKS开式进风隔断阀",
                    阀状态 := "QKS开式进风隔断阀",
                    阀开报警 := "AKS开式进风隔断阀开报警",
                    阀关报警 := "AKS开式进风隔断阀关报警");


           #闭式进风隔断阀(模式设定 := "PW".MS模式设定,
                    条件1 := 0.0,
                    条件2 := 0.0,
                    阀开信号 := "IBS闭式进风隔断阀开反馈",
                    阀关信号 := "IBS闭式进风隔断阀关反馈",
                    手动控制按钮开 := "MBS闭式进风隔断阀",
                    阀状态 := "QBS闭式进风隔断阀",
                    阀开报警 := "ABS闭式进风隔断阀开报警",
                    阀关报警 := "ABS闭式进风隔断阀关报警");

           #一级冷却水阀(模式设定 := "PW".MS模式设定,
                   条件1 := 0.0,
                   条件2 := 0.0,
                   阀开信号 := "IYJ一级冷却水阀开反馈",
                   阀关信号 := "IYJ一级冷却水阀关反馈",
                   手动控制按钮开 := "MYJ一级冷却水阀",
                   阀状态 := "QYJ一级冷却水阀",
                   阀开报警 := "AYJ一级冷却水阀开报警",
                   阀关报警 := "AYJ一级冷却水阀关报警");


           #二级冷冻水阀(模式设定 := "PW".MS模式设定,//Q点不对
                   条件1 := 0.0,
                   条件2 := 0.0,
                   阀开信号 := "IEJ二级冷冻水阀开反馈",
                   阀关信号 := "IEJ二级冷冻水阀关反馈",
                   手动控制按钮开 := "MEJ二级冷冻水阀",
                   阀状态 := "QEJ二级冷冻水阀",
                   阀开报警 := "AEJ二级冷冻水阀开报警",
                   阀关报警 := "AEJ二级冷冻水阀关报警");

           #一级排液阀(模式设定 := "PW".MS模式设定,
                  条件1 := 0.0,
                  条件2 := 0.0,
                  阀开信号 := "IYJ一级排液阀开反馈",
                  阀关信号 := "IYJ一级排液阀关反馈",
                  手动控制按钮开 := "MYJ一级排液阀",
                  阀状态 := "QYJ一级排液阀",
                  阀开报警 := "AYJ一级排液阀开报警",
                  阀关报警 := "AYJ一级排液阀关报警");


           #二级排液阀(模式设定 := "PW".MS模式设定,
                  条件1 := 0.0,
                  条件2 := 0.0,
                  阀开信号 := "IEJ二级排液阀开反馈",
                  阀关信号 := "IEJ二级排液阀关反馈",
                  手动控制按钮开 := "MEJ二级排液阀",
                  阀状态 := "QEJ二级排液阀",
                  阀开报警 := "AEJ二级排液阀开报警",
                  阀关报警 := "AEJ二级排液阀关报警");

           #除雾排液阀(模式设定 := "PW".MS模式设定,
                  条件1 := 0.0,
                  条件2 := 0.0,
                  阀开信号 := "ICW除雾排液阀开反馈",
                  阀关信号 := "ICW除雾排液阀关反馈",
                  手动控制按钮开 := "MCW除雾排液阀",
                  阀状态 := "QCW除雾排液阀",
                  阀开报警 := "ACW除雾排液阀开报警",
                  阀关报警 := "ACW除雾排液阀关报警");

           #补氮阀(模式设定 := "PW".MS模式设定,
                条件1 := 0.0,
                条件2 := 0.0,
                阀开信号 := "IBD补氮阀开反馈",
                阀关信号 := "IBD补氮阀关反馈",
                手动控制按钮开 := "MBD补氮阀",
                阀状态 := "QBD补氮阀",
                阀开报警 := "ABD补氮阀开报警",
                阀关报警 := "ABD补氮阀关报警");

           #进氮阀(模式设定 := "PW".MS模式设定,
                条件1 := 0.0,
                条件2 := 0.0,
                阀开信号 := "IJD进氮阀开反馈",
                阀关信号 := "IJD进氮阀关反馈",
                手动控制按钮开 := "MJD进氮阀",
                阀状态 := "QJD进氮阀",
                阀开报警 := "AJD进氮阀开报警",
                阀关报警 := "AJD进氮阀关报警");


           #塔顶清洗球阀(模式设定 := "PW".MS模式设定,
                   条件1 := 0.0,
                   条件2 := 0.0,
                   阀开信号 := "ITD塔顶清洗球阀开反馈",
                   阀关信号 := "ITD塔顶清洗球阀关反馈",
                   手动控制按钮开 := "MTD塔顶清洗球阀",
                   阀状态 := "QTD塔顶清洗球阀",
                   阀开报警 := "ATD塔顶清洗球阀开报警",
                   阀关报警 := "ATD塔顶清洗球阀关报警");

           #溶剂回收排放阀(模式设定 := "PW".MS模式设定,
                    条件1 := 0.0,
                    条件2 := 0.0,
                    阀开信号 := "IRJ溶剂回收排放阀开反馈",
                    阀关信号 := "IRJ溶剂回收排放阀关反馈",
                    手动控制按钮开 := "MRJ溶剂回收排放阀",
                    阀状态 := "QRJ溶剂回收排放阀",
                    阀开报警 := "ARJ溶剂回收排放阀开报警",
                    阀关报警 := "ARJ溶剂回收排放阀关报警");


           #室内排水隔膜泵(模式设定 := "PW".MS模式设定,
                    条件1 := 0.0,
                    条件2 := 0.0,
                    阀开信号 := "ISN室内排水开反馈",
                    阀关信号 := "ISN室内排水关反馈",
                    手动控制按钮开 := "MSN室内排水隔膜泵",
                    阀状态 := "QSN室内排水隔膜泵",
                    阀开报警 := "ASN室内排水开反馈报警",
                    阀关报警 := "ASN室内排水关反馈报警");


           #溶剂排液泵(模式设定 := "PW".MS模式设定,
                  条件1 := 0.0,
                  条件2 := 0.0,
                  阀开信号 := "IRJ溶剂排液泵开反馈",
                  阀关信号 := "IRJ溶剂排液泵关反馈",
                  手动控制按钮开 := "MRJ溶剂排液泵",
                  阀状态 := "QRJ溶剂排液泵",
                  阀开报警 :="ARJ溶剂排液泵开报警" ,
                  阀关报警 := "ARJ溶剂排液泵关报警");



         (*  #清洗伸缩气缸(模式设定 := "PW".MS模式设定,
                  条件1 := 0.0,
                  条件2 := 0.0,
                  阀开信号 := "IQX清洗伸缩气缸开反馈",
                  阀关信号 := "IQX清洗伸缩气缸关反馈",

                  阀状态 := "QQG气缸升降阀",
                  阀开报警 := "AQX清洗伸缩气缸开报警",
                  阀关报警 := "AQX清洗伸缩气缸关报警"); *)


   END_REGION
END_FUNCTION_BLOCK

FUNCTION_BLOCK "A3-普通阀控制"   // FB7, SCL
{ S7_Optimized_Access := 'TRUE' }
VERSION : 0.1
// stored: AutoNumber true, IsIECCheckEnabled false, IsRetainMemResEnabled false, MemoryReserve 100, SetENOAutomatically false, UDAEnableTagReadback false
   VAR_INPUT
      模式设定 : Real;
      条件1 : Real;
      条件2 : Real;
      阀开信号 : Bool;
      阀关信号 : Bool;
   END_VAR
   VAR_IN_OUT
      手动控制按钮开 : Bool;
      阀状态 : Bool;
      阀开报警 : Bool;
      阀关报警 : Bool;
   END_VAR
   VAR
      TON1 : TON_TIME;
      TON2 { S7_SetPoint := 'True'} : TON_TIME;
   END_VAR
BEGIN
   //手动控制--------------------------------------------------------------------------------------------------------------
   IF #模式设定 = 2.0 OR #模式设定 = 3.0 OR #模式设定 = 4.0  OR #模式设定 = 5.0  OR #模式设定 = 6.0 THEN
       IF #手动控制按钮开 THEN
           #阀状态 := TRUE;
       ELSE
           #阀状态 := FALSE;
       END_IF;
   END_IF;

   #TON1(IN := #"阀状态" AND NOT #"阀开信号",
         PT := T#10s,
         Q => #"阀开报警");
   IF NOT #"阀状态" THEN

       #"阀开报警" := FALSE;
   END_IF;


   #TON2(IN := #"阀状态" = FALSE AND NOT #"阀关信号",
         PT := T#10s,
         Q => #"阀关报警");
   IF #"阀状态" THEN

       #"阀关报警" := FALSE;
   END_IF;
END_FUNCTION_BLOCK

FUNCTION_BLOCK "A4-脉冲控制"   // FB11, SCL
{ S7_Optimized_Access := 'TRUE' }
VERSION : 0.1
// stored: AutoNumber true, IsIECCheckEnabled false, IsRetainMemResEnabled false, MemoryReserve 100, SetENOAutomatically false, UDAEnableTagReadback false
   VAR
      主塔气锤 { S7_SetPoint := 'True'} : "A3-脉冲轮询";
      二级旋风振打锤 { S7_SetPoint := 'True'} : "A3-脉冲轮询";
      一级旋风振打锤 { S7_SetPoint := 'True'} : "A3-脉冲轮询";
      一级旋风振荡器 { S7_SetPoint := 'True'} : "A3-脉冲轮询";
      布袋气锤 { S7_SetPoint := 'True'} : "A3-脉冲轮询";
      布袋反吹 { S7_SetPoint := 'True'} : "A3-脉冲轮询";
      设备振打 { S7_SetPoint := 'True'} : "A3-脉冲轮询";
      输送出料 { S7_SetPoint := 'True'} : "A3-脉冲轮询";
      布袋出料 { S7_SetPoint := 'True'} : "A3-脉冲轮询";
      一级旋风出料 { S7_SetPoint := 'True'} : "A3-脉冲轮询";
      二级旋风出料 { S7_SetPoint := 'True'} : "A3-脉冲轮询";
      布袋出料1 { S7_SetPoint := 'True'} : "A9-循环下料控制";
      一级旋风出料1 { S7_SetPoint := 'True'} : "A9-循环下料控制";
      二级旋风出料1 { S7_SetPoint := 'True'} : "A9-循环下料控制";
      LT1 : Real := 5.0;
   END_VAR
BEGIN
   REGION 脉冲控制
       #一级旋风振打锤(num:=1,
                On_Time:=0.2,
                output_1=>"QYJ一级旋风振打锤",
                Stop_Time:="SV".YJ一级旋风振打间隔,
                脉冲开关:="MYJ一级旋风振打锤");

       #二级旋风振打锤(num := 1,
                On_Time := 0.2,
                output_1 => "QEJ二级旋风振打锤",
                Stop_Time:="SV".EJ二级旋风振打间隔,
                脉冲开关 := "MEJ二级旋风振打锤");

       #一级旋风振荡器(num := 1,
                On_Time := "SV".YJ一级旋风振荡运行,
                output_1 => "QYJ一级旋风振荡器",
                Stop_Time := "SV".YJ一级旋风振荡停止,
                脉冲开关 := "MYJ一级旋风振荡器");


       #主塔气锤(num := 4,
              On_Time := 0.2,
              output_1 => "QZT主塔气锤1",
              output_2 => "QZT主塔气锤2",
              output_3 => "QZT主塔气锤3",
              output_4 => "QZT主塔气锤4",
              Stop_Time := "SV".ZT主塔振打间隔,
              脉冲开关 := "MZT主塔气锤");

       #布袋气锤(num := 2,
              On_Time := 0.2,
              output_1 => "QCC除尘气锤1",
              output_2 => "QCC除尘气锤2",
              Stop_Time := "SV".BD布袋振打时间,
              脉冲开关 := "MCC除尘气锤");

       (* #布袋反吹(num := 2,
              On_Time := 0.2,
              output_1 => "QCC除尘气锤1",
              output_2 => "QCC除尘气锤2",
              Stop_Time := "SV".BD布袋振打时间,
              脉冲开关 := "MCC除尘气锤"); *)

        #设备振打(num := 1,
              On_Time := 0.2,
              output_1 => "QSB设备振打",
              Stop_Time := "SV".SB设备振打间隔,
              脉冲开关 := "MSB设备振打");



        (* #输送出料(num := 2,
              On_Time := 0.2,
              output_1 => "QCC除尘气锤1",
              output_2 => "QCC除尘气锤2",
              Stop_Time := "SV".BD布袋振打时间,
              脉冲开关 := "MCC除尘气锤"); *)

   (*     #布袋出料(num := 2,
              On_Time := "SV".BD布袋T出料设定,
              output_1 => "MCC除尘出料上阀",
              output_2 => "MCC除尘出料下阀",
              Stop_Time := "SV".BD布袋出料设定,
              脉冲开关 := "MBD布袋出料");

        #一级旋风出料(num := 2,
                On_Time := "SV".YJ一级旋风T出料设定,
              output_1 => "MYJ一级出料上阀",
              output_2 => "MYJ一级出料下阀",
              Stop_Time := "SV".YJ一级旋风出料设定,
              脉冲开关 := "MYJ一级出料");

      #二级旋风出料(num := 2,
              On_Time :="SV".EJ二级旋风T出料设定,
              output_1 => "MEJ二级出料上阀",
              output_2 => "MEJ二级出料下阀",
              Stop_Time :="SV".EJ二级旋风出料设定 ,
              脉冲开关 := "MEJ二级出料"); *)


        IF "PW".MS模式设定 = 1.0 OR "PW".MS模式设定 = 3.0 THEN

            #布袋出料1(下料启动开关 := "MBD布袋出料",
                   上卸料阀工作时间 := "SV".BD布袋上阀开时间,
                   上卸料阀关闭时间 := "SV".BD布袋上阀关时间,
                   下卸料阀工作时间 := "SV".BD布袋下阀开时间,
                   下卸料阀关闭时间 := "SV".BD布袋下阀关时间,
                   上下料阀 := "MCC除尘出料上阀",
                   下下料阀 := "MCC除尘出料下阀");


            #一级旋风出料1(下料启动开关 := "MYJ一级出料",
                     上卸料阀工作时间 := "SV".YJ一级旋风上阀开时间,
                     上卸料阀关闭时间 := "SV".YJ一级旋风上阀关时间,
                     下卸料阀工作时间 := "SV".YJ一级旋风下阀开时间,
                     下卸料阀关闭时间 := "SV".YJ一级旋风下阀关时间,
                     上下料阀 := "MYJ一级出料上阀",
                     下下料阀 := "MYJ一级出料下阀");

            #二级旋风出料1(下料启动开关 := "MEJ二级出料",
                     上卸料阀工作时间 := "SV".EJ二级旋风上阀开时间,
                     上卸料阀关闭时间 := "SV".EJ二级旋风上阀关时间,
                     下卸料阀工作时间 := "SV".EJ二级旋风下阀开时间,
                     下卸料阀关闭时间 := "SV".EJ二级旋风下阀关时间,
                     上下料阀 := "MEJ二级出料上阀",
                     下下料阀 := "MEJ二级出料下阀");

        END_IF;


   END_REGION
END_FUNCTION_BLOCK

FUNCTION_BLOCK "A3-脉冲轮询"   // FB12, SCL
{ S7_Optimized_Access := 'TRUE' }
VERSION : 0.1
// stored: AutoNumber true, IsIECCheckEnabled false, IsRetainMemResEnabled false, MemoryReserve 100, SetENOAutomatically false, UDAEnableTagReadback false
   VAR_INPUT
      num : Int;
      On_Time : Real;
   END_VAR
   VAR_OUTPUT
      output_1 : Bool;
      output_2 : Bool;
      output_3 : Bool;
      output_4 : Bool;
      output_5 : Bool;
      output_6 : Bool;
      output_7 : Bool;
      output_8 : Bool;
      output_9 : Bool;
      output_10 : Bool;
      output_11 : Bool;
      output_12 : Bool;
      output_13 : Bool;
      output_14 : Bool;
      output_15 : Bool;
      output_16 : Bool;
   END_VAR
   VAR_IN_OUT
      Stop_Time : Real;
      脉冲开关 : Bool;
      i : Int;
   END_VAR
   VAR
      t1 : TON_TIME;
      t2 { S7_SetPoint := 'True'} : TON_TIME;
      TM_FZ { ExternalAccessible := 'False'; ExternalVisible := 'False'; ExternalWritable := 'False'} : Bool;
      j : Int;
      output_ : Array[0..16] of Bool;
   END_VAR
   VAR RETAIN
      out_ : Array[0..16] of Bool;
   END_VAR
   VAR
      间隔时间 : Time := T#5s;
      运行时间 : Time := T#5s;
   END_VAR
   VAR_TEMP
      "m" : Int;
   END_VAR
BEGIN

   #间隔时间 := DINT_TO_TIME(REAL_TO_DINT(#Stop_Time * 1000.0));
   #运行时间 := DINT_TO_TIME(REAL_TO_DINT(#On_Time * 1000));


   #t1(IN := (1 <> #TM_FZ) AND #脉冲开关,
       PT := #间隔时间);

   #t2(IN := (1 = #TM_FZ) AND #脉冲开关,
       PT := #运行时间);

   IF #t1.Q THEN
       #TM_FZ := 1;
       #output_[#i] := 1;
   END_IF;

   IF #t2.Q THEN
       #TM_FZ := 0;
       #output_[#i] := 0;
       #i += 1;

   END_IF;

   IF #i >= #num OR #i < 0 OR (NOT #脉冲开关) THEN
       #i := 0;
       #TM_FZ := 0;
       FOR #j := 0 TO #num DO
           #output_[#j] := 0;
           IF (#j >= #num)
           THEN
               EXIT;
           END_IF;
       END_FOR;
   END_IF;


   FOR #m := 0 TO 16 DO
       IF #output_[#m] = TRUE THEN
           #out_[#m] := TRUE;
       ELSE
           #out_[#m] := FALSE;
       END_IF;
   END_FOR;
   #output_1 := #out_[0];
   #output_2 := #out_[1];
   #output_3 := #out_[2];
   #output_4 := #out_[3];
   #output_5 := #out_[4];
   #output_6 := #out_[5];
   #output_7 := #out_[6];
   #output_8 := #out_[7];
   #output_9 := #out_[8];
   #output_10 := #out_[9];

   #output_11 := #out_[10];
   #output_12 := #out_[11];
   #output_13 := #out_[12];
   #output_14 := #out_[13];
   #output_15 := #out_[14];
   #output_16 := #out_[15];
END_FUNCTION_BLOCK

FUNCTION_BLOCK "A9-循环下料控制"   // FB15, SCL
{ S7_Optimized_Access := 'TRUE' }
VERSION : 0.1
// stored: AutoNumber true, IsIECCheckEnabled false, IsRetainMemResEnabled false, MemoryReserve 100, SetENOAutomatically false, UDAEnableTagReadback false
   VAR_INPUT
      下料启动开关 : Bool;
      上卸料阀工作时间 : Real;
      上卸料阀关闭时间 : Real;
      下卸料阀工作时间 : Real;
      下卸料阀关闭时间 : Real;
   END_VAR
   VAR_OUTPUT
      上阀实际工作时间 : Real;
      上阀实际停止时间 : Real;
      下阀实际工作时间 : Real;
      下阀实际停止时间 : Real;
   END_VAR
   VAR_IN_OUT
      上下料阀 : Bool;
      下下料阀 : Bool;
      振动筛 : Bool;
   END_VAR
   VAR
      上下料阀实际工作时间 : Time;
      上下料阀实际停止时间 : Time;
      下下料阀实际工作时间 : Time;
      下下料阀实际停止时间 : Time;
      循环间隔实际时间 : Time;
      上阀打开辅助 : Bool;
      上阀关闭辅助 : Bool;
      下阀打开辅助 : Bool;
      下阀关闭辅助 : Bool;
      循环工作时间延时 { S7_SetPoint := 'True'} : TON_TIME;
      上阀打开检测1 { S7_SetPoint := 'True'} : R_TRIG;
      上阀打开检测2 { S7_SetPoint := 'True'} : R_TRIG;
      上阀工作时间延时 { S7_SetPoint := 'True'} : TON_TIME;
      上阀停止时间延时 { S7_SetPoint := 'True'} : TON_TIME;
      下阀工作时间延时 { S7_SetPoint := 'True'} : TON_TIME;
      下阀停止时间延时 { S7_SetPoint := 'True'} : TON_TIME;
      下阀打开检测 { S7_SetPoint := 'True'} : R_TRIG;
   END_VAR
BEGIN

   #上下料阀实际工作时间 := DINT_TO_TIME(REAL_TO_DINT(#上卸料阀工作时间*1000.0));
   #上下料阀实际停止时间 := DINT_TO_TIME(REAL_TO_DINT(#上卸料阀关闭时间 * 1000.0));
   #下下料阀实际工作时间 := DINT_TO_TIME(REAL_TO_DINT(#下卸料阀工作时间 * 1000.0));
   #下下料阀实际停止时间 := DINT_TO_TIME(REAL_TO_DINT(#下卸料阀关闭时间 * 1000.0));

   #上阀打开检测1(CLK:=#下料启动开关);


   IF #上阀打开检测1.Q THEN
       #上阀打开辅助 := TRUE;
   END_IF;


   #上阀工作时间延时.TON(IN:=#上阀打开辅助 AND #下料启动开关 AND NOT #下阀停止时间延时.Q,PT:=#上下料阀实际工作时间);

   #上阀停止时间延时.TON(IN:=#上阀工作时间延时.Q,PT:=#上下料阀实际停止时间);

   #下阀工作时间延时(IN:=#上阀工作时间延时.Q AND #上阀停止时间延时.Q,PT:=#下下料阀实际工作时间);

   #下阀停止时间延时(IN :=#上阀工作时间延时.Q AND #上阀停止时间延时.Q AND  #下阀工作时间延时.Q,PT := #下下料阀实际停止时间);

   #下阀打开检测(CLK:=#下下料阀);


   #上下料阀 := #上阀打开辅助 AND NOT #上阀工作时间延时.Q AND #下料启动开关;


   #下下料阀 := #上阀工作时间延时.Q AND #上阀停止时间延时.Q AND NOT #下阀工作时间延时.Q AND #下料启动开关;

   IF #下阀打开检测.Q AND #下料启动开关 THEN
       #振动筛 := true;
   END_IF;

   IF NOT #下料启动开关 THEN
       #上阀打开辅助 := false;
   END_IF;

   IF #上下料阀 THEN
       #上阀实际工作时间 := DINT_TO_REAL(TIME_TO_DINT(#上阀工作时间延时.ET))/1000.0;
   END_IF;

   IF #上阀工作时间延时.Q AND NOT #上阀停止时间延时.Q THEN
       #上阀实际停止时间 := DINT_TO_REAL(TIME_TO_DINT(#上阀停止时间延时.ET)) / 1000.0;
   END_IF;

   IF #下下料阀 THEN
       #下阀实际工作时间 := DINT_TO_REAL(TIME_TO_DINT(#下阀工作时间延时.ET)) / 1000.0;
   END_IF;

   IF #下阀工作时间延时.Q AND NOT #下阀停止时间延时.Q THEN
       #下阀实际停止时间 := DINT_TO_REAL(TIME_TO_DINT(#下阀停止时间延时.ET)) / 1000.0;
   END_IF;
END_FUNCTION_BLOCK

FUNCTION_BLOCK "R_TRIG"   // FB1001, SCL
AUTHOR : SIMATIC
FAMILY : BIT
NAME : R_TRIG
VERSION : 1.0
// stored: IsIECCheckEnabled false, SetENOAutomatically false, UDAEnableTagReadback false
   VAR_INPUT
      CLK : Bool;   // Input bit
   END_VAR
   VAR_OUTPUT
      Q : Bool;   // Edge detection
   END_VAR
   VAR
      Stat_Bit : Bool;   // edge memory bit used to store the previous signal state
   END_VAR
BEGIN
END_FUNCTION_BLOCK

FUNCTION_BLOCK "A5-模拟量输出"   // FB29, SCL
{ S7_Optimized_Access := 'TRUE' }
VERSION : 0.1
// stored: AutoNumber true, IsIECCheckEnabled false, IsRetainMemResEnabled false, MemoryReserve 100, SetENOAutomatically false, UDAEnableTagReadback false
   VAR
      进风加热比例调节阀 { S7_SetPoint := 'True'} : "A2-数据转换RTI";
      回风加热比例调节阀 { S7_SetPoint := 'True'} : "A2-数据转换RTI";
      放空比例调节阀 { S7_SetPoint := 'True'} : "A2-数据转换RTI";
   END_VAR
BEGIN
   REGION 模拟量输出
       #进风加热比例调节阀(I_Max := 27648,
                  I_Min := 5530,
                  R_Max := 100.0,
                  R_Min := 0.0,
                  R_Value := "SV".JF进风加热比例调节阀,
                  I_ChValue => "QWJF进风加热比例调节阀");

       #回风加热比例调节阀(I_Max := 27648,
                  I_Min := 5530,
                  R_Max := 100.0,
                  R_Min := 0.0,
                  R_Value := "SV".HF回风加热比例调节阀,
                  I_ChValue => "QWHF回风加热比例调节阀");

       #放空比例调节阀(I_Max := 27648,
                I_Min := 5530,
                R_Max := 100.0,
                R_Min := 0.0,
                R_Value := "SV".FK放空比例调节阀,
                I_ChValue => "QWFK放空比例调节阀");
   END_REGION
END_FUNCTION_BLOCK

FUNCTION_BLOCK "A2-数据转换RTI"   // FB48, SCL
{ S7_Optimized_Access := 'TRUE' }
VERSION : 0.1
// stored: AutoNumber true, IsIECCheckEnabled false, IsRetainMemResEnabled false, MemoryReserve 100, SetENOAutomatically false, UDAEnableTagReadback false
   VAR_INPUT
      I_Max : Int := 27648;
      I_Min : Int := 0;
      R_Max : Real;
      R_Min : Real;
      R_Value : Real;
   END_VAR
   VAR_OUTPUT
      I_ChValue : Int;
   END_VAR
BEGIN
   (**)
   #I_ChValue := REAL_TO_INT((#R_Value - #R_Min) / (#R_Max - #R_Min) *( #I_Max-#I_Min))+#I_Min;
   (* OUT = [((FLOAT (IN) – K1)/(K2–K1)) * (HI_LIM–LO_LIM)] + LO_LIM *)
END_FUNCTION_BLOCK

FUNCTION_BLOCK "B1--ALARM"   // FB71, SCL
{ S7_Optimized_Access := 'TRUE' }
VERSION : 0.1
// stored: AutoNumber true, IsIECCheckEnabled false, IsRetainMemResEnabled false, MemoryReserve 100, SetENOAutomatically false, UDAEnableTagReadback false
   VAR
      报警列表1 { S7_SetPoint := 'True'} : "A8-报警功能块";
      报警列表2 { S7_SetPoint := 'True'} : "A8-报警功能块";
      报警列表3 { S7_SetPoint := 'True'} : "A8-报警功能块";
      报警列表4 { S7_SetPoint := 'True'} : "A8-报警功能块";
      报警列表5 { S7_SetPoint := 'True'} : "A8-报警功能块";
      报警列表6 { S7_SetPoint := 'True'} : "A8-报警功能块";
      报警列表7 { S7_SetPoint := 'True'} : "A8-报警功能块";
      报警列表8 { S7_SetPoint := 'True'} : "A8-报警功能块";
      报警列表9 { S7_SetPoint := 'True'} : "A8-报警功能块";
      报警列表10 { S7_SetPoint := 'True'} : "A8-报警功能块";
      报警列表11 { S7_SetPoint := 'True'} : "A8-报警功能块";
      报警列表12 { S7_SetPoint := 'True'} : "A8-报警功能块";
      报警列表13 { S7_SetPoint := 'True'} : "A8-报警功能块";
   END_VAR
BEGIN
   #报警列表1(报警0:="ABD布袋压差低报",
          报警1:="ABD布袋压差变送器故障",
          报警2:="ABD布袋压差高报",
          报警3:="ABD布袋压差高高报",
          报警4:="ABD补氮阀关报警",
          报警5:="ABD补氮阀开报警",
          报警6:="ABP爆破片1反馈报警",
          报警7:="ABP爆破片2反馈报警",
          报警8:="ABS闭式排风隔断阀关报警",
          报警9:="ABS闭式排风隔断阀开报警",
          报警10:="ABS闭式进风隔断阀关报警",
          报警11:="ABS闭式进风隔断阀开报警",
          报警12:="ACC除尘出料上阀关报警",
          报警13:="ACC除尘出料上阀开报警",
          报警14:="ACC除尘出料下阀关报警",
          报警15:="ACC除尘出料下阀开报警");

   #报警列表2(报警0:="ACF出风压差变送器故障",
          报警1:="ACF出风温度故障",
          报警2:="ACF出风温度过低",
          报警3:="ACF出风温度高报",
          报警4:="ACF出风温度高高报",
          报警5:="ACF出风高效低报",
          报警6:="ACF出风高效高报",
          报警7:="ACF出风高效高高报",
          报警8:="ACW除雾排液阀关报警",
          报警9:="ACW除雾排液阀开报警",
          报警10:="ACW除雾液位计高报",
          报警11:="ACW除雾液位计高高报",
          报警12:="ACW除雾溶剂液位计故障",
          报警13:="ADJ电加热报警",
          报警14:="A备用报警1",
          报警15:="AEJ二级冷冻水阀关报警");

   #报警列表3(报警0:="AEJ二级冷冻水阀开报警",
          报警1:="AEJ二级出料上阀关报警",
          报警2:="AEJ二级出料上阀开报警",
          报警3:="AEJ二级出料下阀关报警",
          报警4:="AEJ二级出料下阀开报警",
          报警5:="AEJ二级排液阀关报警",
          报警6:="AEJ二级排液阀开报警",
          报警7:="AEJ二级液位计高报",
          报警8:="AEJ二级液位计高高报",
          报警9:="AEJ二级溶剂液位计故障",
          报警10:="AFD阀导气压低低报",
          报警11:="AFD阀导气压低报",
          报警12:="AFD阀岛气压低低报",
          报警13:="AFD阀岛气压低报",
          报警14:="AFD阀岛气压故障报警",
          报警15:="AFK放空比例反馈故障");

   #报警列表4(报警0:="AGD管道压力变送器故障",
          报警1:="AGD管道压力高报",
          报警2:="AGD管道压力高高报",
          报警3:="AHF回风加热比例反馈故障",
          报警4:="AHF回风温度故障报警",
          报警5:="AHF回风温度高报",
          报警6:="AHF回风温度高高报",
          报警7:="AHS回收罐1报警",
          报警8:="AHS回收罐2报警",
          报警9:="AJB搅拌电机报警",
          报警10:="AJD进氮压力低低报",
          报警11:="AJD进氮压力低报",
          报警12:="AJD进氮压力故障",
          报警13:="AJD进氮阀关报警",
          报警14:="AJD进氮阀开报警",
          报警15:="AJF进风保护温度报警");

   #报警列表5(报警0:="AJF进风冷却水流量低报警",
          报警1:="AJF进风冷却水阀关报警",
          报警2:="AJF进风冷却水阀开报警",
          报警3:="AJF进风加热比例反馈故障",
          报警4:="AJF进风压差低报",
          报警5:="AJF进风压差变送器故障",
          报警6:="AJF进风压差高报",
          报警7:="AJF进风压差高高报",
          报警8:="AJF进风流量低低报",
          报警9:="AJF进风流量低报",
          报警10:="AJF进风流量计故障",
          报警11:="AJF进风温度故障",
          报警12:="AJF进风温度高报",
          报警13:="AJF进风温度高高报",
          报警14:="AJL进料压力故障",
          报警15:="AJL进料压力高报");

   #报警列表6(报警0:="AJL进料压力高高报",
          报警1:="AJL进料泵故障报警",
          报警2:="AJL进料流量低低报",
          报警3:="AJL进料流量低报",
          报警4:="AJL进料流量故障",
          报警5:="AJT急停报警",
          报警6:="AJX机械温控故障",
          报警7:="AKS开式排风隔断阀关报警",
          报警8:="AKS开式排风隔断阀开报警",
          报警9:="AKS开式进风隔断阀关报警",
          报警10:="AKS开式进风隔断阀开报警",
          报警11:="AKY空压低压信号",
          报警12:="ALD冷冻水关报警",
          报警13:="ALD冷冻水流量低报警",
          报警14:="ALQ冷却水流量低报警",
          报警15:="ALX离心雾化故障");

   #报警列表7(报警0:="APY排液流量低报警",
          报警1:="AQL气流雾化阀关报警",
          报警2:="AQL气流雾化阀开报警",
          报警3:="AQT气体检测低低报",
          报警4:="AQT气体检测低报",
          报警5:="AQX清洗伸缩气缸关报警",
          报警6:="AQX清洗伸缩气缸开报警",
          报警7:="AQZ前置液位低低报",
          报警8:="AQZ前置液位低报",
          报警9:="AQZ前置液位计故障",
          报警10:="ARJ溶剂回收排放阀关报警",
          报警11:="ARJ溶剂回收排放阀开报警",
          报警12:="ASF输送加热故障报警",
          报警13:="ASF输送风机故障报警",
          报警14:="ASF输送高效低报",
          报警15:="ASF送风机报警");

   #报警列表8(报警0:="ASN室内排水关反馈报警",
          报警1:="ASN室内排水开反馈报警",
          报警2:="ASS输送保护温度报警",
          报警3:="ASS输送出料上阀关报警",
          报警4:="ASS输送出料上阀开报警",
          报警5:="ASS输送出料下阀关报警",
          报警6:="ASS输送出料下阀开报警",
          报警7:="ASS输送加热报警",
          报警8:="ASS输送温度故障报警",
          报警9:="ASS输送温度高报",
          报警10:="ASS输送温度高高报",
          报警11:="ASS输送进风阀关报警",
          报警12:="ASS输送进风阀开报警",
          报警13:="ASS输送高效低报",
          报警14:="ASS输送高效压差变送器故障",
          报警15:="ASS输送高效高报");

   #报警列表9(报警0:="ASS输送高效高高报",
          报警1:="ATD塔顶清洗球阀关报警",
          报警2:="ATD塔顶清洗球阀开报警",
          报警3:="ATN塔内压力低低报",
          报警4:="ATN塔内压力低报",
          报警5:="ATN塔内压力故障",
          报警6:="ATN塔内压力高报",
          报警7:="ATN塔内压力高高报",
          报警8:="AWH雾化关报警",
          报警9:="AWH雾化开报警",
          报警10:="AWH雾化油压低低报",
          报警11:="AWH雾化油压低报",
          报警12:="AWH雾化油压故障",
          报警13:="AWH雾化进氮低报",
          报警14:="AWK温控未通信",
          报警15:="AWK温控高温报警");

   #报警列表10(报警0:="AWQ尾气故障",
           报警1:="AWQ尾气温度高报",
           报警2:="AWQ尾气温度高高报",
           报警3:="AXY泄压阀关报警",
           报警4:="AXY泄压阀开报警",
           报警5:="AYF引风机报警",
           报警6:="AYH氧含仪1故障",
           报警7:="AYH氧含仪2故障",
           报警8:="AYH氧含仪高报",
           报警9:="AYH氧含仪高高报",
           报警10:="AYH氧含量运行故障",
           报警11:="AYJ一级冷却水阀关报警",
           报警12:="AYJ一级冷却水阀开报警",
           报警13:="AYJ一级出料上阀关报警",
           报警14:="AYJ一级出料上阀开报警",
           报警15:="AYJ一级出料下阀关报警");

   #报警列表11(报警0:="AYJ一级出料下阀开报警",
           报警1:="AYJ一级排液阀关报警",
           报警2:="AYJ一级排液阀开报警",
           报警3:="AYJ一级液位计高报",
           报警4:="AYJ一级液位计高高报",
           报警5:="AYJ一级溶剂液位计故障",
           报警6:="AKS开式自动自检不通过",
           报警7:="ACIP缺水报警",
           报警8:="ARJ溶剂排液泵开报警",
           报警9:="ARJ溶剂排液泵关报警");
END_FUNCTION_BLOCK

FUNCTION_BLOCK "A8-报警功能块"   // FB13, SCL
{ S7_Optimized_Access := 'TRUE' }
VERSION : 0.1
// stored: AutoNumber true, IsIECCheckEnabled false, IsRetainMemResEnabled false, MemoryReserve 100, SetENOAutomatically false, UDAEnableTagReadback false
   VAR_INPUT
      报警0 : Bool;
      报警1 : Bool;
      报警2 : Bool;
      报警3 : Bool;
      报警4 : Bool;
      报警5 : Bool;
      报警6 : Bool;
      报警7 : Bool;
      报警8 : Bool;
      报警9 : Bool;
      报警10 : Bool;
      报警11 : Bool;
      报警12 : Bool;
      报警13 : Bool;
      报警14 : Bool;
      报警15 : Bool;
   END_VAR
   VAR
      报警 : Word;
      报警文本 : Array[0..15] of WString[20];
      off : Bool;
   END_VAR
BEGIN
    IF NOT  #off THEN

           #报警文本[0] := GetSymbolName(variable := #报警0, size := 0);
           #报警文本[1] := GetSymbolName(variable := #报警1, size := 0);
           #报警文本[2] := GetSymbolName(variable := #报警2, size := 0);
           #报警文本[3] := GetSymbolName(variable := #报警3, size := 0);
           #报警文本[4] := GetSymbolName(variable := #报警4, size := 0);
           #报警文本[5] := GetSymbolName(variable := #报警5, size := 0);
           #报警文本[6] := GetSymbolName(variable := #报警6, size := 0);
           #报警文本[7] := GetSymbolName(variable := #报警7, size := 0);

           #报警文本[8] := GetSymbolName(variable := #报警8, size := 0);
           #报警文本[9] := GetSymbolName(variable := #报警9, size := 0);
           #报警文本[10] := GetSymbolName(variable := #报警10, size := 0);
           #报警文本[11] := GetSymbolName(variable := #报警11, size := 0);
           #报警文本[12] := GetSymbolName(variable := #报警12, size := 0);
           #报警文本[13] := GetSymbolName(variable := #报警13, size := 0);
           #报警文本[14] := GetSymbolName(variable := #报警14, size := 0);
           #报警文本[15] := GetSymbolName(variable := #报警15, size := 0);

       END_IF;

       IF #报警0 THEN
           #报警.%X0 := 1;
       ELSE
           #报警.%X0 := 0;
       END_IF;

       IF #报警1 THEN
           #报警.%X1 := 1;
       ELSE
           #报警.%X1 := 0;
       END_IF;

       IF #报警2 THEN
           #报警.%X2 := 1;
       ELSE
           #报警.%X2 := 0;
       END_IF;


       IF #报警3 THEN
           #报警.%X3 := 1;
       ELSE
           #报警.%X3 := 0;
       END_IF;

       IF #报警4 THEN
           #报警.%X4 := 1;
       ELSE
           #报警.%X4 := 0;
       END_IF;

       IF #报警5 THEN
           #报警.%X5 := 1;
       ELSE
           #报警.%X5 := 0;
       END_IF;

       IF #报警6 THEN
           #报警.%X6 := 1;
       ELSE
           #报警.%X6 := 0;
       END_IF;

       IF #报警7 THEN
           #报警.%X7 := 1;
       ELSE
           #报警.%X7 := 0;
       END_IF;



       IF #报警8 THEN
           #报警.%X8 := 1;
       ELSE
           #报警.%X8 := 0;
       END_IF;

       IF #报警9 THEN
           #报警.%X9 := 1;
       ELSE
           #报警.%X9 := 0;
       END_IF;

       IF #报警10 THEN
           #报警.%X10 := 1;
       ELSE
           #报警.%X10 := 0;
       END_IF;


       IF #报警11 THEN
           #报警.%X11 := 1;
       ELSE
           #报警.%X11 := 0;
       END_IF;

       IF #报警12 THEN
           #报警.%X12 := 1;
       ELSE
           #报警.%X12 := 0;
       END_IF;

       IF #报警13 THEN
           #报警.%X13 := 1;
       ELSE
           #报警.%X13 := 0;
       END_IF;

       IF #报警14 THEN
           #报警.%X14 := 1;
       ELSE
           #报警.%X14 := 0;
       END_IF;

       IF #报警15 THEN
           #报警.%X15 := 1;
       ELSE
           #报警.%X15 := 0;
       END_IF;
END_FUNCTION_BLOCK

FUNCTION_BLOCK "B4-清洗连锁"   // FB58, SCL
{ S7_Optimized_Access := 'TRUE' }
VERSION : 0.1
// stored: AutoNumber true, IsIECCheckEnabled false, IsRetainMemResEnabled false, MemoryReserve 100, SetENOAutomatically false, UDAEnableTagReadback false
   VAR
      TON0 : TON_TIME;
      TON1 : TON_TIME;
      TON2 { S7_SetPoint := 'True'} : TON_TIME;
      TON3 { S7_SetPoint := 'True'} : TON_TIME;
      TON4 { S7_SetPoint := 'True'} : TON_TIME;
      TON5 { S7_SetPoint := 'True'} : TON_TIME;
      TON6 { S7_SetPoint := 'True'} : TON_TIME;
      TON7 { S7_SetPoint := 'True'} : TON_TIME;
      R_TRIG { S7_SetPoint := 'True'} : Array[0..100] of R_TRIG;
      RT { S7_SetPoint := 'True'} : Array[0..100] of Bool;
      F_TRIG { S7_SetPoint := 'True'} : Array[0..100] of F_TRIG;
      FT { S7_SetPoint := 'True'} : Array[0..100] of Bool;
      BJ报警上升辅助 : Bool;
      BJ报警下降辅助 : Bool;
      BJ报警上升沿 { S7_SetPoint := 'True'} : R_TRIG;
      BJ报警下降沿 { S7_SetPoint := 'True'} : F_TRIG;
      F1 { S7_SetPoint := 'True'} : Bool;
      F2 : Bool;
      ET0 : Time;
      ET1 : Time;
      ET2 : Time;
      ET3 : Time;
      ET4 : Time;
      ET5 : Time;
      ET6 : Time;
      ET7 : Time;
      F3 : Bool;
      F4 : Bool;
      Temp_1 : Int;
      AERROR : Bool;
      t0_1s : TON_TIME;
      YC1 { S7_SetPoint := 'True'} : DInt;
      YC2 : DInt;
      YC3 : DInt;
      YC4 : DInt;
      YC5 : DInt;
   END_VAR
BEGIN
   IF "PW".MS模式设定 = 5.0 OR "PW".MS模式设定 = 6.0 OR "PW".MS模式设定 = 2.0 THEN

       IF "MFZ仿真调试" THEN
           IF "QQG气缸升" = 0 AND "QQG气缸降" = 1 THEN
               "IQX清洗伸缩气缸降反馈" := 1;
           END_IF;

           IF "QQG气缸升" = 1 AND "QQG气缸降" = 0 THEN
               "IQX清洗伸缩气缸升反馈" := 1;
           END_IF;

          (* IF "MQG气缸升" THEN
               "QQG气缸升" := 1;
           ELSE
               "QQG气缸升" := 0;
           END_IF;

           IF "MQG气缸降" THEN
               "QQG气缸降" := 1;
           ELSE
               "QQG气缸降" := 0;
           END_IF; *)

       END_IF;




       IF "ATD塔顶清洗球阀开报警" OR "ATD塔顶清洗球阀关报警" THEN
           #AERROR := 1;
       ELSE
           #AERROR := 0;
       END_IF;

       IF "MZT主塔伸缩气缸" THEN
           "MQG气缸升" := 0;
           "QQG气缸升" := 0;
           "MQG气缸降" := 1;
           "QQG气缸降" := 1;
       ELSE
           "MQG气缸升" := 1;
           "QQG气缸升" := 1;
           "MQG气缸降" := 0;
           "QQG气缸降" := 0;

       END_IF;


      (* #TON1(IN := "MTD塔顶清洗阀" AND NOT #AERROR,
             PT := T#5s,
             ET => #ET1);

       #TON2(IN := "MZT主塔伸缩气缸" AND #"QQ气缸下限位" AND NOT #AERROR AND "MTD塔顶清洗阀",
             PT := T#5s,
             ET => #ET2); *)

       IF "MZT主塔清洗"  THEN
           #YC3 := 0;
           #YC4 := 0;

           "MTD塔顶清洗球阀" := 1;
           "QTD塔顶清洗球阀" := 1;

           IF "QTD塔顶清洗球阀" AND #t0_1s.Q AND #YC1 < 10 THEN
               #YC1 := #YC1 + 1;
           END_IF;

           IF #YC1 >= 10.0 THEN
               "MZT主塔伸缩气缸" := 1;
               #YC1 := 0;
           END_IF;

           IF "IQX清洗伸缩气缸降反馈" AND #t0_1s.Q AND #YC2 < 10 THEN
               #YC2 := #YC2 + 1;
           END_IF;

           IF #YC2 >= 10 AND "MZT主塔清洗进水阀" THEN
               "MZT主塔清洗进水阀" := 1;
               "QZT主塔清洗进水阀" := 1;
               //"MTD塔顶清洗阀" := 1;
              // "QTD塔顶清洗阀" := 1;
           END_IF;
       END_IF;


       IF NOT "MZT主塔清洗" THEN
           #YC1 := 0;
           #YC2 := 0;
          // "MTD塔顶清洗阀" := 0;
          // "QTD塔顶清洗阀" := 0;
           "MZT主塔清洗进水阀" := 0;
           "QZT主塔清洗进水阀" := 0;

           IF NOT "QZT主塔清洗进水阀"  AND #t0_1s.Q AND #YC3 < 10 THEN
               #YC3 := #YC3 + 1;
           END_IF;

           IF #YC3 >= 10.0 AND NOT "QZT主塔清洗进水阀"  THEN
               "MZT主塔伸缩气缸" := 0;

           END_IF;

           IF "IQX清洗伸缩气缸升反馈" AND #t0_1s.Q AND #YC4 < 10 THEN
               #YC4 := #YC4 + 1;
           END_IF;

           IF #YC4 >= 10 AND "IQX清洗伸缩气缸升反馈" THEN
               "MTD塔顶清洗球阀" := 0;
               "QTD塔顶清洗球阀" := 0;
               #YC3 := 0;
               #YC4 := 0;
           END_IF;

       END_IF;

   END_IF;

   #t0_1s(IN := NOT #t0_1s.Q,
          PT := t#1000ms);
END_FUNCTION_BLOCK

FUNCTION_BLOCK "F_TRIG"   // FB1002, SCL
AUTHOR : SIMATIC
FAMILY : BIT
NAME : F_TRIG
VERSION : 1.0
// stored: IsIECCheckEnabled false, SetENOAutomatically false, UDAEnableTagReadback false
   VAR_INPUT
      CLK : Bool;   // Input bit
   END_VAR
   VAR_OUTPUT
      Q : Bool;   // Edge detection
   END_VAR
   VAR
      Stat_Bit : Bool;   // edge memory bit used to store the previous signal state
   END_VAR
BEGIN
END_FUNCTION_BLOCK

FUNCTION "0- IO Configure" : Void   // FC10, LAD
TITLE = 1_IO Configure
{ S7_Optimized_Access := 'TRUE' }
VERSION : 0.1
// stored: AutoNumber true, IsIECCheckEnabled false, SetENOAutomatically false, UDAEnableTagReadback false
BEGIN

REGION Network 1 (SCL): IJT急停
   //DI/DO地址分配-----------------------------------------------------------------------
   //"SV".JF进风加热比例调节阀
   //"MYH氧含仪隔断阀"
   //"AWQ尾气温度高高报"
   //"AYJ一级排液阀开报警"



   "ISF送风机" := NOT "I0.0";
   "IYF引风机" := NOT "I0.1";
   "ILX离心雾化器" := NOT "I0.2";
   "IJL进料泵" := "I0.3";
   "IDJ电加热" :=  "I0.4";
   "ISF输送风机" := "I0.5";
   "ISF输送加热" := "I0.6";
   "IJT急停" := "I0.7";

   "ILQ冷却水流量" := "I1.0";
   "ILD冷冻水流量" := "I1.1";
   "IJF进风冷却水流量" := "I1.2";
   "IPY排液流量" := "I1.3";
   "IBD补氮阀开反馈" := "I1.4";
   "IBD补氮阀关反馈" := "I1.5";
   "IJD进氮阀开反馈" := "I1.6";
   "IJD进氮阀关反馈" := "I1.7";

   "IXY泄压阀开反馈" := "I2.0";
   "IXY泄压阀关反馈" := "I2.1";
   "IQL气流雾化阀开反馈" := "I2.2";
   "IQL气流雾化阀关反馈" := "I2.3";
   "ISF输送进风阀开反馈" := "I2.4";
   "ISF输送进风阀关反馈" := "I2.5";
   "IKS开式排风隔断阀开反馈" := "I2.6";
   "IKS开式排风隔断阀关反馈" := "I2.7";

   "IBS闭式排风隔断阀开反馈" := "I3.0";
   "IBS闭式排风隔断阀关反馈" := "I3.1";
   "IKS开式进风隔断阀开反馈" := "I3.2";
   "IKS开式进风隔断阀关反馈" := "I3.3";
   "IBS闭式进风隔断阀开反馈" := "I3.4";
   "IBS闭式进风隔断阀关反馈" := "I3.5";
   "IYJ一级冷却水阀开反馈" := "I3.6";
   "IYJ一级冷却水阀关反馈" := "I3.7";

   "IEJ二级冷冻水阀开反馈" := "I4.0";
   "IEJ二级冷冻水阀关反馈" := "I4.1";
   "IYJ一级排液阀开反馈" := "I4.2";
   "IYJ一级排液阀关反馈" := "I4.3";
   "IEJ二级排液阀开反馈" := "I4.4";
   "IEJ二级排液阀关反馈" := "I4.5";
   "ICW除雾排液阀开反馈" := "I4.6";
   "ICW除雾排液阀关反馈" := "I4.7";

   "IRJ溶剂回收排放阀开反馈" := "I5.0";
   "IRJ溶剂回收排放阀关反馈" := "I5.1";
   "IJF进风冷却水阀开反馈" := "I5.3";
   "IJF进风冷却水阀关反馈" := "I5.2";

   "ITD塔顶清洗球阀开反馈" := "I5.4";
   "ITD塔顶清洗球阀关反馈" := "I5.5";

   "IQX清洗伸缩气缸升反馈" := "I5.6";//升
   "IQX清洗伸缩气缸降反馈" := "I5.7";//降

   "IJF进风保护温度" := "I6.0";
   "ISS输送保护温度" := "I6.1";
   "IBP爆破片1反馈" := NOT "I6.2";
   "IBP爆破片2反馈" := NOT "I6.3";
   "ISN室内排水开反馈" := "I6.7";
   "ISN室内排水关反馈" := "I6.6";
   "IRJ溶剂排液泵开反馈" := "I6.4";
   "IRJ溶剂排液泵关反馈" := "I6.5";

   (* 冷却水流量开关报警
   冷冻水流量开关报警
   进风冷却水流量开关报警
   排液流量开关报警
    电加热故障
   输送风机故障
   输送加热故障
   爆破片1故障
   爆破片2故障

   *)
   "AQX清洗伸缩气缸关报警" := 0;
   "AQX清洗伸缩气缸开报警" := 0;

   (* IF "ILQ冷却水流量" THEN
       "ALQ冷却水流量低报警" := 1;
   ELSE
       "ALQ冷却水流量低报警" := 0;
   END_IF;

   IF "ILD冷冻水流量" THEN
       "ALD冷冻水流量低报警" := 1;
   ELSE
       "ALD冷冻水流量低报警" := 0;
   END_IF; *)

   IF "IJF进风冷却水流量" THEN
       "AJF进风冷却水流量低报警" := 1;
   ELSE
       "AJF进风冷却水流量低报警" := 0;
   END_IF;

   //暂时注销掉
   (* IF "IPY排液流量" THEN
       "APY排液流量低报警" := 1;
   ELSE
       "APY排液流量低报警" := 0;
   END_IF; *)

   IF "IBP爆破片1反馈" THEN
       "ABP爆破片1反馈报警" := 1;
   ELSE
       "ABP爆破片1反馈报警" := 0;
   END_IF;

   IF "IBP爆破片2反馈" THEN
       "ABP爆破片2反馈报警" := 1;
   ELSE
       "ABP爆破片2反馈报警" := 0;
   END_IF;

   IF "IDJ电加热" THEN
       "ADJ电加热报警" := 1;
   ELSE
       "ADJ电加热报警" := 0;
   END_IF;

   IF "ISF输送风机" THEN
       "ASF输送风机故障报警" := 1;
   ELSE
       "ASF输送风机故障报警" := 0;
   END_IF;


   IF "ISF输送加热" THEN
       "ASF输送加热故障报警" := 1;
   ELSE
       "ASF输送加热故障报警" := 0;
   END_IF;

   IF NOT "IJT急停" THEN
       "AJT急停报警" := 1;
   ELSE
       "AJT急停报警" := 0;
   END_IF;
   (* IF ILQ冷却水流量开关
   冷冻水流量开关报警
   进风冷却水流量开关报警
   排液流量开关报警
   电加热故障
   输送风机故障
   输送加热故障
   爆破片1故障
   爆破片2故障 *)

   "Q0.0" := "QSF送风机";
   "Q0.1" := "QSF送风机风扇";
   "Q0.2" := "QYF引风机";
   "Q0.3" := "QYF引风机风扇";
   "Q0.4" := "QLX离心雾化";
   "Q0.5" := "QLX离心雾化风扇";
   "Q0.6" := "QLX离心雾化油泵";
   "Q0.7" := "QJL进料泵";

   "Q1.0" := "QJL进料泵风扇";
   "Q1.1" := "QDJ电加热器";
   "Q1.2" := "QSS输送风机";
   "Q1.3" := "QSS输送加热器";
   "Q1.4" := "QFM蜂鸣器";
   "Q1.5" := "QZS指示灯";
   "Q1.6" := "QYS钥匙开关";
   "Q1.7" := "QZM照明灯";

   "Q2.0" := "QBY备用1";
   "Q2.1" := "QCC除尘脉冲";
   "Q2.2" := "QBY备用2";
   "Q2.3" := "QBY备用3";
   "Q2.4" := "QBY备用4";
   "Q2.5" := "QRS热水洗请求";
   "Q2.6" := 0;//无
   "Q2.7" := "QBY备用7";

   "Q3.0" := "QXY泄压阀";
   "Q3.1" := "QJF进风冷却水阀";
   "Q3.2" := "QSS输送进风阀";
   "Q3.3" := "QQL气流雾化阀";
   "Q3.4" := "QKS开式排风隔断阀";
   "Q3.5" := "QBS闭式排风隔断阀";
   "Q3.6" := "QKS开式进风隔断阀";
   "Q3.7" := "QBS闭式进风隔断阀";

   "Q4.0" := "QYJ一级冷却水阀";
   "Q4.1" := "QEJ二级冷冻水阀";
   "Q4.2" := "QYJ一级排液阀";
   "Q4.3" := "QEJ二级排液阀";
   "Q4.4" := "QCW除雾排液阀";
   "Q4.5" := "QRJ溶剂回收排放阀";
   "Q4.6" := "QSN室内排水隔膜泵";//回程泵
   "Q4.7" := "QRJ溶剂排液泵";

   "Q5.0" := "QBY备用10";;
   "Q5.1" := "QBY备用11";;
   "Q5.2" := "QASA室内回水阀";//振打
   "Q5.3" := "QBD补氮阀";
   "Q5.4" := "QASA室外回水阀";//振打
   "Q5.5" := "QJD进氮阀";
   "Q5.6" := "QCC除尘气锤1";
   "Q5.7" := "QCC除尘气锤2";

   "Q6.0" := "QTD塔顶清洗球阀";//加阀岛
   "Q6.1" := "QRJ溶剂排液泵进阀";
   "Q6.3" := "QSB设备振打";
   //阀导
   "Q10.0" := "QSN室内清洗总阀"; //室内清洗总阀
   "Q10.1" := "QASA室内回水阀";//A室内回水阀
   "Q10.2" := "QASA室外回水阀";//A室外回水阀
   "Q10.3" := "QJF进风蒸汽开关阀";
   "Q10.4" := "QJF进风蒸汽排水阀";
   "Q10.5" := "QLG料罐清洗阀";
   "Q10.6" := "QQX清洗溶剂出阀";
   "Q10.7" := "QWL物料进阀";

   "Q11.0" := "QYJ一级出料上阀";
   "Q11.1" := "QYJ一级出料下阀";
   "Q11.2" := "QEJ二级出料上阀";
   "Q11.3" := "QEJ二级出料下阀";
   "Q11.4" := "QCC除尘出料上阀";
   "Q11.5" := "QCC除尘出料下阀";
   "Q11.6" := "QHF回风蒸汽开关阀";
   "Q11.7" := "QHF回风蒸汽排水阀";

   "Q12.0" := "QSS输送出料上阀";
   "Q12.1" := "QSS输送出料下阀";//空的，未接
   "Q12.2" := "QQG气缸升";
   "Q12.3" := "QQG气缸降";
   "Q12.4" := "QZT主塔清洗进水阀";
   "Q12.5" := "QXF旋风管道清洗阀";
   "Q12.6" := "QYJ一级旋风清洗阀";
   "Q12.7" := "QEJ二级旋风清洗阀";

